PROGRAM PRG_Governance_Validator_Integrity_Governor
  VAR
    L_Now_MS : UDINT;
    L_Integrity_Valid : BOOL := TRUE;
    L_Error_Code : UDINT := 0;
    L_Error_Text : STRING(160) := '';
  END_VAR

            L_Now_MS := GVL_STATUS.G_System_Time_MS;
L_Integrity_Valid := TRUE;
L_Error_Code := 0;
L_Error_Text := '';

// Fail-safe defaults.
GVL_GOVERNANCE_VALIDATOR_INTEGRITY_FABRIC.Governance_Validator_Integrity_Valid := FALSE;
GVL_GOVERNANCE_VALIDATOR_INTEGRITY_FABRIC.Governance_Validator_Integrity_Granted := FALSE;
GVL_GOVERNANCE_VALIDATOR_INTEGRITY_FABRIC.Governance_Validator_Integrity_Quarantine_Active := TRUE;

GVL_GOVERNANCE_VALIDATOR_INTEGRITY_FABRIC.Validator_Semantics_Immutable := FALSE;
GVL_GOVERNANCE_VALIDATOR_INTEGRITY_FABRIC.CrossEpoch_Validation_Equivalence_Stable := FALSE;
GVL_GOVERNANCE_VALIDATOR_INTEGRITY_FABRIC.Distributed_Validator_Consensus_Valid := FALSE;
GVL_GOVERNANCE_VALIDATOR_INTEGRITY_FABRIC.Governance_Rule_Integrity_Canonical := FALSE;
GVL_GOVERNANCE_VALIDATOR_INTEGRITY_FABRIC.Validator_Lineage_Coherent := FALSE;

// Governance feedback integrity required.
IF NOT GVL_GOVERNANCE_FEEDBACK_INTEGRITY_FABRIC.Governance_Feedback_Integrity_Granted THEN
    L_Integrity_Valid := FALSE;
    L_Error_Code := 53000;
    L_Error_Text := 'Governance feedback integrity not granted';
END_IF;

// Validator self-corruption detectors.
IF GVL_GOVERNANCE_VALIDATOR_INTEGRITY_FABRIC.Validator_Semantic_Drift_Detected THEN
    L_Integrity_Valid := FALSE;
    L_Error_Code := 53001;
    L_Error_Text := 'Validator semantic drift detected';
END_IF;

IF GVL_GOVERNANCE_VALIDATOR_INTEGRITY_FABRIC.CrossNode_Validation_Fork THEN
    L_Integrity_Valid := FALSE;
    L_Error_Code := 53002;
    L_Error_Text := 'Cross-node validation fork detected';
END_IF;

IF GVL_GOVERNANCE_VALIDATOR_INTEGRITY_FABRIC.Governance_Rule_Mutation_Detected THEN
    L_Integrity_Valid := FALSE;
    L_Error_Code := 53003;
    L_Error_Text := 'Governance rule mutation detected';
END_IF;

IF GVL_GOVERNANCE_VALIDATOR_INTEGRITY_FABRIC.SelfReferential_Validator_Corruption THEN
    L_Integrity_Valid := FALSE;
    L_Error_Code := 53004;
    L_Error_Text := 'Self-referential validator corruption detected';
END_IF;

IF GVL_GOVERNANCE_VALIDATOR_INTEGRITY_FABRIC.Validator_Lineage_Drift_Detected THEN
    L_Integrity_Valid := FALSE;
    L_Error_Code := 53005;
    L_Error_Text := 'Validator lineage drift detected';
END_IF;

IF GVL_GOVERNANCE_VALIDATOR_INTEGRITY_FABRIC.Distributed_Validator_Reality_Fork_Detected THEN
    L_Integrity_Valid := FALSE;
    L_Error_Code := 53006;
    L_Error_Text := 'Distributed validator reality fork detected';
END_IF;

// Validator integrity validation.
IF L_Integrity_Valid
AND NOT GVL_GOVERNANCE_VALIDATOR_INTEGRITY_FABRIC.Validator_Causality_Grounded THEN
    L_Integrity_Valid := FALSE;
    L_Error_Code := 53010;
    L_Error_Text := 'Validator causality invalid';
END_IF;

IF L_Integrity_Valid
AND NOT GVL_GOVERNANCE_VALIDATOR_INTEGRITY_FABRIC.Governance_Rule_Evolution_Governed THEN
    L_Integrity_Valid := FALSE;
    L_Error_Code := 53011;
    L_Error_Text := 'Governance rule evolution invalid';
END_IF;

IF L_Integrity_Valid
AND NOT GVL_GOVERNANCE_VALIDATOR_INTEGRITY_FABRIC.Distributed_Validation_Timeline_Monotonic THEN
    L_Integrity_Valid := FALSE;
    L_Error_Code := 53012;
    L_Error_Text := 'Distributed validation timeline monotonicity invalid';
END_IF;

IF L_Integrity_Valid
AND NOT GVL_GOVERNANCE_VALIDATOR_INTEGRITY_FABRIC.Validator_Interpretation_Equivalence_Valid THEN
    L_Integrity_Valid := FALSE;
    L_Error_Code := 53013;
    L_Error_Text := 'Validator interpretation equivalence invalid';
END_IF;

IF L_Integrity_Valid THEN
    GVL_GOVERNANCE_VALIDATOR_INTEGRITY_FABRIC.Governance_Validator_Integrity_Valid := TRUE;
    GVL_GOVERNANCE_VALIDATOR_INTEGRITY_FABRIC.Governance_Validator_Integrity_Granted := TRUE;
    GVL_GOVERNANCE_VALIDATOR_INTEGRITY_FABRIC.Governance_Validator_Integrity_Quarantine_Active := FALSE;

    GVL_GOVERNANCE_VALIDATOR_INTEGRITY_FABRIC.Validator_Semantics_Immutable := TRUE;
    GVL_GOVERNANCE_VALIDATOR_INTEGRITY_FABRIC.CrossEpoch_Validation_Equivalence_Stable := TRUE;
    GVL_GOVERNANCE_VALIDATOR_INTEGRITY_FABRIC.Distributed_Validator_Consensus_Valid := TRUE;
    GVL_GOVERNANCE_VALIDATOR_INTEGRITY_FABRIC.Governance_Rule_Integrity_Canonical := TRUE;
    GVL_GOVERNANCE_VALIDATOR_INTEGRITY_FABRIC.Validator_Lineage_Coherent := TRUE;

    GVL_GOVERNANCE_VALIDATOR_INTEGRITY_FABRIC.Governance_Validator_Integrity_Epoch :=
        GVL_GOVERNANCE_FEEDBACK_INTEGRITY_FABRIC.Governance_Feedback_Integrity_Epoch;

    GVL_GOVERNANCE_VALIDATOR_INTEGRITY_FABRIC.Governance_Validator_Integrity_Epoch_Coherent := TRUE;

    GVL_GOVERNANCE_VALIDATOR_INTEGRITY_FABRIC.Governance_Validator_Integrity_Last_Update_MS :=
        L_Now_MS;

    GVL_GOVERNANCE_VALIDATOR_INTEGRITY_FABRIC.Governance_Validator_Integrity_Lease_Expired := FALSE;

    GVL_GOVERNANCE_VALIDATOR_INTEGRITY_FABRIC.Governance_Validator_Integrity_Last_Error_Code := 0;
    GVL_GOVERNANCE_VALIDATOR_INTEGRITY_FABRIC.Governance_Validator_Integrity_Last_Error_Text := '';
ELSE
    GVL_GOVERNANCE_VALIDATOR_INTEGRITY_FABRIC.Governance_Validator_Integrity_Valid := FALSE;
    GVL_GOVERNANCE_VALIDATOR_INTEGRITY_FABRIC.Governance_Validator_Integrity_Granted := FALSE;
    GVL_GOVERNANCE_VALIDATOR_INTEGRITY_FABRIC.Governance_Validator_Integrity_Quarantine_Active := TRUE;

    GVL_GOVERNANCE_VALIDATOR_INTEGRITY_FABRIC.Governance_Validator_Integrity_Lease_Expired := TRUE;

    GVL_GOVERNANCE_VALIDATOR_INTEGRITY_FABRIC.Governance_Validator_Integrity_Last_Error_Code :=
        L_Error_Code;

    GVL_GOVERNANCE_VALIDATOR_INTEGRITY_FABRIC.Governance_Validator_Integrity_Last_Error_Text :=
        L_Error_Text;

    GVL_GOVERNANCE_VALIDATOR_INTEGRITY_FABRIC.Governance_Validator_Integrity_Invalidation_Count :=
        GVL_GOVERNANCE_VALIDATOR_INTEGRITY_FABRIC.Governance_Validator_Integrity_Invalidation_Count + 1;
END_IF;
          
END_PROGRAM

PROGRAM PRG_Heating_Policy_Observer
  VAR
    fbPolicy : FB_Heating_Policy_Observer;
  END_VAR

            fbPolicy(
    VI_Zone_Occupied := GVL_PRESENCE.G_Zone_Occupied,
    VI_Zone_Last_Motion_TS := GVL_PRESENCE.G_Zone_Last_Motion_TS,
    VI_System_Time_MS := GVL_STATUS.G_System_Time_MS,
    VI_Zone_Permanent_Use := GVL_HEATING_POLICY.G_Zone_Permanent_Use,
    VI_Zone_Guest_Preheat := GVL_HEATING_POLICY.G_Zone_Guest_Preheat_Request,
    VI_Behavior_Mode := GVL_MODE.G_Current_Behavior_Mode
);

GVL_HEATING_POLICY.G_Zone_Empty_Duration_MS := fbPolicy.VO_Zone_Empty_Duration_MS;
GVL_HEATING_POLICY.G_Zone_Policy_Class := fbPolicy.VO_Zone_Policy_Class;
GVL_HEATING_POLICY.G_Zone_Target_Adjustment := fbPolicy.VO_Zone_Target_Adjustment;
GVL_HEATING_POLICY.G_Zone_Priority_Bias := fbPolicy.VO_Zone_Priority_Bias;
          
END_PROGRAM

PROGRAM PRG_Time_Service
  VAR
    fbTimebase : FB_System_Timebase;
    fbTime : FB_Time_Service;
  END_VAR

            // Central time update point.
// Must run before PRG_IO_Read and all consumers of GVL_TIME_SERVICE.
fbTimebase();
fbTime();

// Step 4.2 compatibility bridge.
// Legacy consumers of GVL_STATUS.G_System_Time_MS receive the same canonical time.
GVL_STATUS.G_System_Time_MS := GVL_TIME_SERVICE.G_Now_MS;
GVL_STATUS.G_Current_TOD := GVL_TIME_SERVICE.G_Current_TOD;
GVL_STATUS.G_Current_Day := TO_UINT(GVL_TIME_SERVICE.G_Day_Of_Week);
          
END_PROGRAM

PROGRAM PRG_Operator_Semantic_Alignment_Governor
  VAR
    L_Now_MS : UDINT;
    L_Operator_Valid : BOOL := TRUE;
    L_Error_Code : UDINT := 0;
    L_Error_Text : STRING(160) := '';
  END_VAR

            L_Now_MS := GVL_STATUS.G_System_Time_MS;
L_Operator_Valid := TRUE;
L_Error_Code := 0;
L_Error_Text := '';

// Fail-safe defaults.
GVL_OPERATOR_SEMANTIC_ALIGNMENT.Operator_Semantic_Alignment_Valid := FALSE;
GVL_OPERATOR_SEMANTIC_ALIGNMENT.Operator_Semantic_Alignment_Granted := FALSE;
GVL_OPERATOR_SEMANTIC_ALIGNMENT.Operator_Semantic_Alignment_Quarantine_Active := TRUE;

GVL_OPERATOR_SEMANTIC_ALIGNMENT.HMI_Semantic_State_Coherent := FALSE;
GVL_OPERATOR_SEMANTIC_ALIGNMENT.Operator_Recovery_Intent_Aligned := FALSE;
GVL_OPERATOR_SEMANTIC_ALIGNMENT.Alarm_Semantic_Priority_Coherent := FALSE;
GVL_OPERATOR_SEMANTIC_ALIGNMENT.Runtime_Explanation_Coherent := FALSE;
GVL_OPERATOR_SEMANTIC_ALIGNMENT.Authority_State_Human_Visible := FALSE;

// Semantic preservation required.
IF NOT GVL_SEMANTIC_PRESERVATION_FABRIC.Semantic_Preservation_Granted THEN
    L_Operator_Valid := FALSE;
    L_Error_Code := 40000;
    L_Error_Text := 'Semantic preservation authority not granted';
END_IF;

// Human-machine semantic split-brain detectors.
IF GVL_OPERATOR_SEMANTIC_ALIGNMENT.HMI_Semantic_Lag_Detected THEN
    L_Operator_Valid := FALSE;
    L_Error_Code := 40001;
    L_Error_Text := 'HMI semantic lag detected';
END_IF;

IF GVL_OPERATOR_SEMANTIC_ALIGNMENT.Operator_Interpretation_Skew_Detected THEN
    L_Operator_Valid := FALSE;
    L_Error_Code := 40002;
    L_Error_Text := 'Operator interpretation skew detected';
END_IF;

IF GVL_OPERATOR_SEMANTIC_ALIGNMENT.Alarm_Cognition_Mismatch_Detected THEN
    L_Operator_Valid := FALSE;
    L_Error_Code := 40003;
    L_Error_Text := 'Alarm cognition mismatch detected';
END_IF;

IF GVL_OPERATOR_SEMANTIC_ALIGNMENT.Hidden_Authority_State_Detected THEN
    L_Operator_Valid := FALSE;
    L_Error_Code := 40004;
    L_Error_Text := 'Hidden authority state detected';
END_IF;

IF GVL_OPERATOR_SEMANTIC_ALIGNMENT.Semantic_Explanation_Divergence_Detected THEN
    L_Operator_Valid := FALSE;
    L_Error_Code := 40005;
    L_Error_Text := 'Semantic explanation divergence detected';
END_IF;

IF GVL_OPERATOR_SEMANTIC_ALIGNMENT.Human_Recovery_Misunderstanding_Detected THEN
    L_Operator_Valid := FALSE;
    L_Error_Code := 40006;
    L_Error_Text := 'Human recovery misunderstanding detected';
END_IF;

// Operator cognition coherence validation.
IF L_Operator_Valid
AND NOT GVL_OPERATOR_SEMANTIC_ALIGNMENT.Human_Interpretation_Coherent THEN
    L_Operator_Valid := FALSE;
    L_Error_Code := 40010;
    L_Error_Text := 'Human interpretation coherence invalid';
END_IF;

IF L_Operator_Valid
AND NOT GVL_OPERATOR_SEMANTIC_ALIGNMENT.Adaptive_Runtime_Visibility_Valid THEN
    L_Operator_Valid := FALSE;
    L_Error_Code := 40011;
    L_Error_Text := 'Adaptive runtime visibility invalid';
END_IF;

IF L_Operator_Valid
AND NOT GVL_OPERATOR_SEMANTIC_ALIGNMENT.Semantic_Explanation_Fresh THEN
    L_Operator_Valid := FALSE;
    L_Error_Code := 40012;
    L_Error_Text := 'Semantic explanation freshness invalid';
END_IF;

IF L_Operator_Valid
AND NOT GVL_OPERATOR_SEMANTIC_ALIGNMENT.Operator_Action_Context_Aligned THEN
    L_Operator_Valid := FALSE;
    L_Error_Code := 40013;
    L_Error_Text := 'Operator action context alignment invalid';
END_IF;

IF L_Operator_Valid THEN
    GVL_OPERATOR_SEMANTIC_ALIGNMENT.Operator_Semantic_Alignment_Valid := TRUE;
    GVL_OPERATOR_SEMANTIC_ALIGNMENT.Operator_Semantic_Alignment_Granted := TRUE;
    GVL_OPERATOR_SEMANTIC_ALIGNMENT.Operator_Semantic_Alignment_Quarantine_Active := FALSE;

    GVL_OPERATOR_SEMANTIC_ALIGNMENT.HMI_Semantic_State_Coherent := TRUE;
    GVL_OPERATOR_SEMANTIC_ALIGNMENT.Operator_Recovery_Intent_Aligned := TRUE;
    GVL_OPERATOR_SEMANTIC_ALIGNMENT.Alarm_Semantic_Priority_Coherent := TRUE;
    GVL_OPERATOR_SEMANTIC_ALIGNMENT.Runtime_Explanation_Coherent := TRUE;
    GVL_OPERATOR_SEMANTIC_ALIGNMENT.Authority_State_Human_Visible := TRUE;

    GVL_OPERATOR_SEMANTIC_ALIGNMENT.Operator_Alignment_Epoch :=
        GVL_SEMANTIC_PRESERVATION_FABRIC.Semantic_Preservation_Epoch;

    GVL_OPERATOR_SEMANTIC_ALIGNMENT.Operator_Alignment_Epoch_Coherent := TRUE;

    GVL_OPERATOR_SEMANTIC_ALIGNMENT.Operator_Alignment_Last_Update_MS :=
        L_Now_MS;

    GVL_OPERATOR_SEMANTIC_ALIGNMENT.Operator_Alignment_Lease_Expired := FALSE;

    GVL_OPERATOR_SEMANTIC_ALIGNMENT.Operator_Alignment_Last_Error_Code := 0;
    GVL_OPERATOR_SEMANTIC_ALIGNMENT.Operator_Alignment_Last_Error_Text := '';
ELSE
    GVL_OPERATOR_SEMANTIC_ALIGNMENT.Operator_Semantic_Alignment_Valid := FALSE;
    GVL_OPERATOR_SEMANTIC_ALIGNMENT.Operator_Semantic_Alignment_Granted := FALSE;
    GVL_OPERATOR_SEMANTIC_ALIGNMENT.Operator_Semantic_Alignment_Quarantine_Active := TRUE;

    GVL_OPERATOR_SEMANTIC_ALIGNMENT.Operator_Alignment_Lease_Expired := TRUE;

    GVL_OPERATOR_SEMANTIC_ALIGNMENT.Operator_Alignment_Last_Error_Code :=
        L_Error_Code;

    GVL_OPERATOR_SEMANTIC_ALIGNMENT.Operator_Alignment_Last_Error_Text :=
        L_Error_Text;

    GVL_OPERATOR_SEMANTIC_ALIGNMENT.Operator_Alignment_Invalidation_Count :=
        GVL_OPERATOR_SEMANTIC_ALIGNMENT.Operator_Alignment_Invalidation_Count + 1;
END_IF;
          
END_PROGRAM

PROGRAM PRG_Deterministic_Recovery_Path_Governor
  VAR
    L_Now_MS : UDINT;
  END_VAR

            L_Now_MS := GVL_STATUS.G_System_Time_MS;

IF GVL_CROSSDOMAIN_FAILSAFE_CLOSURE_FABRIC.CrossDomain_FailSafe_Closure_Granted
AND NOT GVL_DETERMINISTIC_RECOVERY_PATH_FABRIC.Unsafe_Recovery_Path_Detected
AND NOT GVL_DETERMINISTIC_RECOVERY_PATH_FABRIC.Recovery_Path_Divergence_Detected
AND NOT GVL_DETERMINISTIC_RECOVERY_PATH_FABRIC.Recovery_Causality_Break_Detected
AND NOT GVL_DETERMINISTIC_RECOVERY_PATH_FABRIC.Distributed_Recovery_Fork_Detected THEN

    GVL_DETERMINISTIC_RECOVERY_PATH_FABRIC.Deterministic_Recovery_Path_Valid := TRUE;
    GVL_DETERMINISTIC_RECOVERY_PATH_FABRIC.Deterministic_Recovery_Path_Granted := TRUE;
    GVL_DETERMINISTIC_RECOVERY_PATH_FABRIC.Deterministic_Recovery_Path_Canonical := TRUE;
    GVL_DETERMINISTIC_RECOVERY_PATH_FABRIC.Recovery_Lineage_Causality_Valid := TRUE;
    GVL_DETERMINISTIC_RECOVERY_PATH_FABRIC.Recovery_Physical_Convergence_Stable := TRUE;
    GVL_DETERMINISTIC_RECOVERY_PATH_FABRIC.Recovery_Timeline_Monotonic := TRUE;

    GVL_DETERMINISTIC_RECOVERY_PATH_FABRIC.Deterministic_Recovery_Path_Epoch :=
        GVL_CROSSDOMAIN_FAILSAFE_CLOSURE_FABRIC.CrossDomain_FailSafe_Closure_Epoch;

    GVL_DETERMINISTIC_RECOVERY_PATH_FABRIC.Deterministic_Recovery_Path_Last_Update_MS :=
        L_Now_MS;
END_IF;
          
END_PROGRAM

PROGRAM PRG_Temporal_Causality_Closure_Governor

            IF GVL_DISTRIBUTED_SAFETY_REALITY_CONSENSUS_FABRIC.Distributed_Safety_Reality_Consensus_Granted
AND NOT GVL_TEMPORAL_CAUSALITY_CLOSURE_FABRIC.Temporal_Fork_Detected
AND NOT GVL_TEMPORAL_CAUSALITY_CLOSURE_FABRIC.Stale_Causality_Application_Detected
AND NOT GVL_TEMPORAL_CAUSALITY_CLOSURE_FABRIC.Recovery_Before_Revocation_Detected
AND NOT GVL_TEMPORAL_CAUSALITY_CLOSURE_FABRIC.Distributed_Timeline_Drift_Detected THEN

    GVL_TEMPORAL_CAUSALITY_CLOSURE_FABRIC.Temporal_Causality_Closure_Valid := TRUE;
    GVL_TEMPORAL_CAUSALITY_CLOSURE_FABRIC.Temporal_Causality_Closure_Granted := TRUE;
    GVL_TEMPORAL_CAUSALITY_CLOSURE_FABRIC.Temporal_Causality_Coherent := TRUE;
    GVL_TEMPORAL_CAUSALITY_CLOSURE_FABRIC.Monotonic_Reality_Timeline_Valid := TRUE;
    GVL_TEMPORAL_CAUSALITY_CLOSURE_FABRIC.Recovery_Revocation_Ordering_Valid := TRUE;
END_IF;
          
END_PROGRAM

PROGRAM PRG_Governance_Liveness_Integrity_Governor
  VAR
    L_Now_MS : UDINT;
    L_Integrity_Valid : BOOL := TRUE;
    L_Error_Code : UDINT := 0;
    L_Error_Text : STRING(160) := '';
  END_VAR

            L_Now_MS := GVL_STATUS.G_System_Time_MS;
L_Integrity_Valid := TRUE;
L_Error_Code := 0;
L_Error_Text := '';

// Fail-safe defaults.
GVL_GOVERNANCE_LIVENESS_INTEGRITY_FABRIC.Governance_Liveness_Integrity_Valid := FALSE;
GVL_GOVERNANCE_LIVENESS_INTEGRITY_FABRIC.Governance_Liveness_Integrity_Granted := FALSE;
GVL_GOVERNANCE_LIVENESS_INTEGRITY_FABRIC.Governance_Liveness_Integrity_Quarantine_Active := TRUE;

GVL_GOVERNANCE_LIVENESS_INTEGRITY_FABRIC.Governance_Execution_Liveness_Stable := FALSE;
GVL_GOVERNANCE_LIVENESS_INTEGRITY_FABRIC.Integrity_Governor_Scheduling_Canonical := FALSE;
GVL_GOVERNANCE_LIVENESS_INTEGRITY_FABRIC.CrossGovernor_Execution_Continuity_Valid := FALSE;
GVL_GOVERNANCE_LIVENESS_INTEGRITY_FABRIC.Deterministic_Validation_Cycle_Integrity := FALSE;
GVL_GOVERNANCE_LIVENESS_INTEGRITY_FABRIC.Governance_Runtime_Liveness_Coherent := FALSE;

// Governance validator integrity required.
IF NOT GVL_GOVERNANCE_VALIDATOR_INTEGRITY_FABRIC.Governance_Validator_Integrity_Granted THEN
    L_Integrity_Valid := FALSE;
    L_Error_Code := 54000;
    L_Error_Text := 'Governance validator integrity not granted';
END_IF;

// Governance liveness degradation detectors.
IF GVL_GOVERNANCE_LIVENESS_INTEGRITY_FABRIC.Integrity_Governor_Starvation_Detected THEN
    L_Integrity_Valid := FALSE;
    L_Error_Code := 54001;
    L_Error_Text := 'Integrity governor starvation detected';
END_IF;

IF GVL_GOVERNANCE_LIVENESS_INTEGRITY_FABRIC.Validation_Cycle_Skip_Detected THEN
    L_Integrity_Valid := FALSE;
    L_Error_Code := 54002;
    L_Error_Text := 'Validation cycle skip detected';
END_IF;

IF GVL_GOVERNANCE_LIVENESS_INTEGRITY_FABRIC.CrossGovernor_Execution_Jitter_Fork THEN
    L_Integrity_Valid := FALSE;
    L_Error_Code := 54003;
    L_Error_Text := 'Cross-governor execution jitter fork detected';
END_IF;

IF GVL_GOVERNANCE_LIVENESS_INTEGRITY_FABRIC.Selective_Governance_Degradation_Detected THEN
    L_Integrity_Valid := FALSE;
    L_Error_Code := 54004;
    L_Error_Text := 'Selective governance degradation detected';
END_IF;

IF GVL_GOVERNANCE_LIVENESS_INTEGRITY_FABRIC.Runtime_Governor_Execution_Stall_Detected THEN
    L_Integrity_Valid := FALSE;
    L_Error_Code := 54005;
    L_Error_Text := 'Runtime governor execution stall detected';
END_IF;

IF GVL_GOVERNANCE_LIVENESS_INTEGRITY_FABRIC.Distributed_Liveness_Reality_Fork_Detected THEN
    L_Integrity_Valid := FALSE;
    L_Error_Code := 54006;
    L_Error_Text := 'Distributed liveness reality fork detected';
END_IF;

// Governance liveness validation.
IF L_Integrity_Valid
AND NOT GVL_GOVERNANCE_LIVENESS_INTEGRITY_FABRIC.Validation_Cycle_Timing_Monotonic THEN
    L_Integrity_Valid := FALSE;
    L_Error_Code := 54010;
    L_Error_Text := 'Validation cycle timing invalid';
END_IF;

IF L_Integrity_Valid
AND NOT GVL_GOVERNANCE_LIVENESS_INTEGRITY_FABRIC.Distributed_Governor_Execution_Aligned THEN
    L_Integrity_Valid := FALSE;
    L_Error_Code := 54011;
    L_Error_Text := 'Distributed governor execution alignment invalid';
END_IF;

IF L_Integrity_Valid
AND NOT GVL_GOVERNANCE_LIVENESS_INTEGRITY_FABRIC.Runtime_Integrity_Causality_Grounded THEN
    L_Integrity_Valid := FALSE;
    L_Error_Code := 54012;
    L_Error_Text := 'Runtime integrity causality invalid';
END_IF;

IF L_Integrity_Valid
AND NOT GVL_GOVERNANCE_LIVENESS_INTEGRITY_FABRIC.Governance_Execution_Budget_Stable THEN
    L_Integrity_Valid := FALSE;
    L_Error_Code := 54013;
    L_Error_Text := 'Governance execution budget invalid';
END_IF;

IF L_Integrity_Valid THEN
    GVL_GOVERNANCE_LIVENESS_INTEGRITY_FABRIC.Governance_Liveness_Integrity_Valid := TRUE;
    GVL_GOVERNANCE_LIVENESS_INTEGRITY_FABRIC.Governance_Liveness_Integrity_Granted := TRUE;
    GVL_GOVERNANCE_LIVENESS_INTEGRITY_FABRIC.Governance_Liveness_Integrity_Quarantine_Active := FALSE;

    GVL_GOVERNANCE_LIVENESS_INTEGRITY_FABRIC.Governance_Execution_Liveness_Stable := TRUE;
    GVL_GOVERNANCE_LIVENESS_INTEGRITY_FABRIC.Integrity_Governor_Scheduling_Canonical := TRUE;
    GVL_GOVERNANCE_LIVENESS_INTEGRITY_FABRIC.CrossGovernor_Execution_Continuity_Valid := TRUE;
    GVL_GOVERNANCE_LIVENESS_INTEGRITY_FABRIC.Deterministic_Validation_Cycle_Integrity := TRUE;
    GVL_GOVERNANCE_LIVENESS_INTEGRITY_FABRIC.Governance_Runtime_Liveness_Coherent := TRUE;

    GVL_GOVERNANCE_LIVENESS_INTEGRITY_FABRIC.Governance_Liveness_Integrity_Epoch :=
        GVL_GOVERNANCE_VALIDATOR_INTEGRITY_FABRIC.Governance_Validator_Integrity_Epoch;

    GVL_GOVERNANCE_LIVENESS_INTEGRITY_FABRIC.Governance_Liveness_Integrity_Epoch_Coherent := TRUE;

    GVL_GOVERNANCE_LIVENESS_INTEGRITY_FABRIC.Governance_Liveness_Integrity_Last_Update_MS :=
        L_Now_MS;

    GVL_GOVERNANCE_LIVENESS_INTEGRITY_FABRIC.Governance_Liveness_Integrity_Lease_Expired := FALSE;

    GVL_GOVERNANCE_LIVENESS_INTEGRITY_FABRIC.Governance_Liveness_Integrity_Last_Error_Code := 0;
    GVL_GOVERNANCE_LIVENESS_INTEGRITY_FABRIC.Governance_Liveness_Integrity_Last_Error_Text := '';
ELSE
    GVL_GOVERNANCE_LIVENESS_INTEGRITY_FABRIC.Governance_Liveness_Integrity_Valid := FALSE;
    GVL_GOVERNANCE_LIVENESS_INTEGRITY_FABRIC.Governance_Liveness_Integrity_Granted := FALSE;
    GVL_GOVERNANCE_LIVENESS_INTEGRITY_FABRIC.Governance_Liveness_Integrity_Quarantine_Active := TRUE;

    GVL_GOVERNANCE_LIVENESS_INTEGRITY_FABRIC.Governance_Liveness_Integrity_Lease_Expired := TRUE;

    GVL_GOVERNANCE_LIVENESS_INTEGRITY_FABRIC.Governance_Liveness_Integrity_Last_Error_Code :=
        L_Error_Code;

    GVL_GOVERNANCE_LIVENESS_INTEGRITY_FABRIC.Governance_Liveness_Integrity_Last_Error_Text :=
        L_Error_Text;

    GVL_GOVERNANCE_LIVENESS_INTEGRITY_FABRIC.Governance_Liveness_Integrity_Invalidation_Count :=
        GVL_GOVERNANCE_LIVENESS_INTEGRITY_FABRIC.Governance_Liveness_Integrity_Invalidation_Count + 1;
END_IF;
          
END_PROGRAM

PROGRAM PRG_Runtime_Compression_Governor

            // ARCHITECTURAL CONSOLIDATION & RUNTIME COMPRESSION
// READ-ONLY / NON-INVASIVE

GVL_CANONICAL_RUNTIME_FABRIC_REGISTRY.Runtime_Complexity_Pressure_Observed :=
    GVL_SURVIVABILITY_INTELLIGENCE_FABRIC.Governance_Saturation_Pressure_Observed;

GVL_CANONICAL_RUNTIME_FABRIC_REGISTRY.Governance_Runtime_Cost_Observed :=
    GVL_OPERATIONAL_INTELLIGENCE_FABRIC.Governance_Complexity_Pressure_Observed;

GVL_CANONICAL_RUNTIME_FABRIC_REGISTRY.Verification_Induced_Instability_Risk :=
    GVL_SURVIVABILITY_INTELLIGENCE_FABRIC.Chronic_Degradation_Risk_Increasing;

IF GVL_OPERATIONAL_INTELLIGENCE_FABRIC.Governance_Saturation_Observed THEN
    GVL_CANONICAL_RUNTIME_FABRIC_REGISTRY.Governance_Scattering_Observed := TRUE;
    GVL_CANONICAL_RUNTIME_FABRIC_REGISTRY.Semantic_Duplication_Observed := TRUE;
END_IF;

IF GVL_CANONICAL_RUNTIME_FABRIC_REGISTRY.Runtime_Complexity_Pressure_Observed THEN
    GVL_CANONICAL_RUNTIME_FABRIC_REGISTRY.Governance_Depth_Limit_Reached := TRUE;
END_IF;

IF GVL_CANONICAL_RUNTIME_FABRIC_REGISTRY.Governance_Runtime_Cost_Observed THEN
    GVL_CANONICAL_RUNTIME_FABRIC_REGISTRY.Verification_Chaining_Limit_Reached := TRUE;
END_IF;

IF GVL_OPERATIONAL_INTELLIGENCE_FABRIC.Operational_Opacity_Observed THEN
    GVL_CANONICAL_RUNTIME_FABRIC_REGISTRY.Observability_Amplification_Limit_Reached := TRUE;
END_IF;
          
END_PROGRAM

PROGRAM PRG_Distributed_Runtime_Supervisor
  VAR
    fbClusterSafetyBarrier : FB_Cluster_Safety_Barrier_Runtime;
    fbRuntimeDiscovery : FB_Runtime_Node_Discovery;
    fbRuntimeSessions : FB_Runtime_Session_Governance;
    fbDistributedRuntimeContinuity : FB_Distributed_Runtime_Continuity;
    fbDistributedAuthority : FB_Distributed_Authority_Arbitration;
    fbRuntimeBusReplication : FB_Runtime_Bus_Replication;
    fbMQTTRuntimeAdapter : FB_MQTT_Runtime_Adapter;
    fbOPCUARuntimeAdapter : FB_OPCUA_Runtime_Adapter;
    fbADSRuntimeAdapter : FB_ADS_Runtime_Adapter;
    fbProjectionOwnership : FB_Distributed_Projection_Ownership_Runtime;
    fbDistributedOrchestration : FB_Distributed_Orchestration_Runtime;
    fbRecoveryLock : FB_Distributed_Recovery_Lock_Runtime;
    fbExecutionGates : FB_Distributed_Execution_Gates_Runtime;
    fbClusterRuntimeFSM : FB_Cluster_Runtime_FSM;
  END_VAR

            // Root distributed runtime execution chain.
//
// Execution order intentionally deterministic:
// safety -> discovery -> sessions -> authority -> replication
// -> transport -> ownership -> orchestration -> recovery locking
// -> unified execution gates -> cluster runtime FSM.
//
// Important convergence contract:
// execution gates must never reopen distributed execution authority
// before finalized convergence/publication continuity is achieved.
//
// Required finalized authority chain:
// immutable snapshot
// -> distributed reconciliation
// -> distributed commit continuity
// -> finalized publication validity
// -> convergence release
// -> execution gates reopen.

fbClusterSafetyBarrier(
    VI_Enable := TRUE,
    VI_System_Time_MS := GVL_STATUS.G_System_Time_MS
);

fbRuntimeDiscovery(
    VI_Enable := TRUE,
    VI_System_Time_MS := GVL_STATUS.G_System_Time_MS
);

fbRuntimeSessions(
    VI_Enable := TRUE,
    VI_System_Time_MS := GVL_STATUS.G_System_Time_MS
);

fbDistributedRuntimeContinuity(
    VI_Enable := TRUE,
    VI_System_Time_MS := GVL_STATUS.G_System_Time_MS
);

fbDistributedAuthority(
    VI_Enable := TRUE,
    VI_System_Time_MS := GVL_STATUS.G_System_Time_MS
);

fbRuntimeBusReplication(
    VI_Enable := TRUE,
    VI_System_Time_MS := GVL_STATUS.G_System_Time_MS
);

fbMQTTRuntimeAdapter(
    VI_Enable := TRUE,
    VI_System_Time_MS := GVL_STATUS.G_System_Time_MS
);

fbOPCUARuntimeAdapter(
    VI_Enable := TRUE,
    VI_System_Time_MS := GVL_STATUS.G_System_Time_MS
);

fbADSRuntimeAdapter(
    VI_Enable := TRUE,
    VI_System_Time_MS := GVL_STATUS.G_System_Time_MS
);

fbProjectionOwnership(
    VI_Enable := TRUE,
    VI_System_Time_MS := GVL_STATUS.G_System_Time_MS
);

fbDistributedOrchestration(
    VI_Enable := TRUE,
    VI_System_Time_MS := GVL_STATUS.G_System_Time_MS
);

fbRecoveryLock(
    VI_Enable := TRUE,
    VI_System_Time_MS := GVL_STATUS.G_System_Time_MS
);

fbExecutionGates(
    VI_Enable := TRUE,
    VI_System_Time_MS := GVL_STATUS.G_System_Time_MS
);

fbClusterRuntimeFSM(
    VI_Enable := TRUE,
    VI_System_Time_MS := GVL_STATUS.G_System_Time_MS
);
          
END_PROGRAM

PROGRAM PRG_Authority_Lineage_Governor
  VAR
    L_Now_MS : UDINT;
    L_Lineage_Valid : BOOL := TRUE;
    L_Error_Code : UDINT := 0;
    L_Error_Text : STRING(160) := '';
  END_VAR

            L_Now_MS := GVL_STATUS.G_System_Time_MS;
L_Lineage_Valid := TRUE;
L_Error_Code := 0;
L_Error_Text := '';

GVL_AUTHORITY_LINEAGE.Authority_Lineage_Valid := FALSE;
GVL_AUTHORITY_LINEAGE.Warm_Restart_Continuity_Valid := FALSE;
GVL_AUTHORITY_LINEAGE.HA_Resume_Continuity_Valid := FALSE;
GVL_AUTHORITY_LINEAGE.Retained_State_Integrity_Valid := FALSE;

IF GVL_AUTHORITY_LINEAGE.Authority_Replay_Suspected THEN
    L_Lineage_Valid := FALSE;
    L_Error_Code := 25000;
    L_Error_Text := 'Authority replay suspected';
END_IF;

IF L_Lineage_Valid AND GVL_AUTHORITY_LINEAGE.Retained_State_Skew_Detected THEN
    L_Lineage_Valid := FALSE;
    L_Error_Code := 25001;
    L_Error_Text := 'Retained state skew detected';
END_IF;

IF L_Lineage_Valid AND GVL_AUTHORITY_LINEAGE.Partial_Authority_Resurrection_Detected THEN
    L_Lineage_Valid := FALSE;
    L_Error_Code := 25002;
    L_Error_Text := 'Partial authority resurrection detected';
END_IF;

IF L_Lineage_Valid AND GVL_AUTHORITY_LINEAGE.Epoch_Lineage_Discontinuity_Detected THEN
    L_Lineage_Valid := FALSE;
    L_Error_Code := 25003;
    L_Error_Text := 'Epoch lineage discontinuity detected';
END_IF;

IF L_Lineage_Valid
AND (ULINT_TO_UDINT(GVL_PHYSICAL_AUTHORITY_EPOCH.Physical_Authority_Epoch) < GVL_AUTHORITY_LINEAGE.Last_Physical_Authority_Epoch) THEN
    GVL_AUTHORITY_LINEAGE.Authority_Replay_Suspected := TRUE;
    L_Lineage_Valid := FALSE;
    L_Error_Code := 25010;
    L_Error_Text := 'Physical authority epoch rollback detected';
END_IF;

IF L_Lineage_Valid
AND (ULINT_TO_UDINT(GVL_RUNTIME_EPOCH.Runtime_Epoch) < GVL_AUTHORITY_LINEAGE.Last_Runtime_Epoch) THEN
    GVL_AUTHORITY_LINEAGE.Retained_State_Skew_Detected := TRUE;
    L_Lineage_Valid := FALSE;
    L_Error_Code := 25011;
    L_Error_Text := 'Runtime epoch rollback detected';
END_IF;

IF L_Lineage_Valid
AND (ULINT_TO_UDINT(GVL_OUTPUT_EPOCH.Output_Publication_Epoch) < GVL_AUTHORITY_LINEAGE.Last_Output_Publication_Epoch) THEN
    GVL_AUTHORITY_LINEAGE.Partial_Authority_Resurrection_Detected := TRUE;
    L_Lineage_Valid := FALSE;
    L_Error_Code := 25012;
    L_Error_Text := 'Output publication epoch rollback detected';
END_IF;

IF L_Lineage_Valid THEN
    GVL_AUTHORITY_LINEAGE.Authority_Lineage_Valid := TRUE;
    GVL_AUTHORITY_LINEAGE.Warm_Restart_Continuity_Valid := TRUE;
    GVL_AUTHORITY_LINEAGE.HA_Resume_Continuity_Valid := TRUE;
    GVL_AUTHORITY_LINEAGE.Retained_State_Integrity_Valid := TRUE;

    GVL_AUTHORITY_LINEAGE.Authority_Lineage_Epoch := ULINT_TO_UDINT(GVL_PHYSICAL_AUTHORITY_EPOCH.Physical_Authority_Epoch);
    GVL_AUTHORITY_LINEAGE.Last_Physical_Authority_Epoch := ULINT_TO_UDINT(GVL_PHYSICAL_AUTHORITY_EPOCH.Physical_Authority_Epoch);
    GVL_AUTHORITY_LINEAGE.Last_Runtime_Epoch := ULINT_TO_UDINT(GVL_RUNTIME_EPOCH.Runtime_Epoch);
    GVL_AUTHORITY_LINEAGE.Last_Output_Publication_Epoch := ULINT_TO_UDINT(GVL_OUTPUT_EPOCH.Output_Publication_Epoch);
    GVL_AUTHORITY_LINEAGE.Authority_Lineage_Last_Update_MS := L_Now_MS;
    GVL_AUTHORITY_LINEAGE.Authority_Lineage_Last_Error_Code := 0;
    GVL_AUTHORITY_LINEAGE.Authority_Lineage_Last_Error_Text := '';
ELSE
    GVL_AUTHORITY_LINEAGE.Authority_Lineage_Valid := FALSE;
    GVL_AUTHORITY_LINEAGE.Authority_Lineage_Last_Error_Code := L_Error_Code;
    GVL_AUTHORITY_LINEAGE.Authority_Lineage_Last_Error_Text := L_Error_Text;
    GVL_AUTHORITY_LINEAGE.Authority_Lineage_Invalidation_Count := GVL_AUTHORITY_LINEAGE.Authority_Lineage_Invalidation_Count + 1;
END_IF;
          
END_PROGRAM

PROGRAM PRG_System_Alarm_Gateway
  VAR
    fbSystemAlarmOrchestrator : FB_System_Alarm_Orchestrator;
    fbSystemGatewayIntent : FB_System_Gateway_Intent;
    L_Scenario_Req_Gateway : E_SCENARIO_TYPE;
  END_VAR

            // Alarm orchestration based on global health snapshot
fbSystemAlarmOrchestrator(
    VI_First_Fault_Active := GVL_SYSTEM_HEALTH.G_First_Fault_Active,
    VI_First_Fault_Type := GVL_SYSTEM_HEALTH.G_First_Fault_Type,
    VI_First_Fault_Source := GVL_SYSTEM_HEALTH.G_First_Fault_Source
);

// Gateway intent execution
fbSystemGatewayIntent(
    VI_System_Time_MS := GVL_TIME_SERVICE.G_Now_MS,
    VI_IsActivePLC := GVL_STATUS.G_Is_Active_PLC,
    VI_Gateway_Writes_Allowed := NOT GVL_STATUS.G_Diagnostics.Operator_Action_Blocked,
    VIO_FloorHeating_Temps := GVL_STATE.G_Floor_Temps,
    VIO_Zone_Valve_States := GVL_STATE.G_Zone_Valves,
    VIO_Lighting_Base_Levels := GVL_STATE.G_Lighting_Levels,
    VIO_Scenario_Req_Gateway := L_Scenario_Req_Gateway
);

GVL_INTENT_USER.I_Scenario_Request := L_Scenario_Req_Gateway;
          
END_PROGRAM

PROGRAM PRG_Debug_View
  VAR
    L_i : INT;
    L_MaxWeight : REAL;
    L_MinWeight : REAL;
    L_Weight : REAL;
    L_Index : INT;
  END_VAR

            GVL_DEBUG_VIEW.D_Current_Time_MS := GVL_TIME_SERVICE.G_Now_MS;

GVL_DEBUG_VIEW.D_Safety_Mode := GVL_SAFETY_SHUTDOWN.G_Safety_Mode;
GVL_DEBUG_VIEW.D_Safety_Active := (GVL_SAFETY_SHUTDOWN.G_Safety_Mode <> NORMAL);
GVL_DEBUG_VIEW.D_Recovery_Phase := GVL_SAFETY_RECOVERY.G_Recovery_Phase;
GVL_DEBUG_VIEW.D_Recovery_Active := GVL_SAFETY_RECOVERY.G_Recovery_Active;

GVL_DEBUG_VIEW.D_Current_Scenario := GVL_INTENT_BEHAVIOR.I_Selected_Scenario_Text;
GVL_DEBUG_VIEW.D_Behavior_Reason := GVL_INTENT_BEHAVIOR.I_Reason_Text;

GVL_DEBUG_VIEW.D_Score_Night := GVL_INTENT_BEHAVIOR.I_Score_Night;
GVL_DEBUG_VIEW.D_Score_Preheat := GVL_INTENT_BEHAVIOR.I_Score_Preheat;
GVL_DEBUG_VIEW.D_Score_VentBoost := GVL_INTENT_BEHAVIOR.I_Score_Vent_Boost;
GVL_DEBUG_VIEW.D_Score_AccessSecure := GVL_INTENT_BEHAVIOR.I_Score_Access_Secure;

GVL_DEBUG_VIEW.D_Intent_Night := GVL_INTENT_BEHAVIOR.I_Request_Night_Mode;
GVL_DEBUG_VIEW.D_Intent_Comfort := GVL_INTENT_BEHAVIOR.I_Request_Comfort_Mode;
GVL_DEBUG_VIEW.D_Intent_VentBoost := GVL_INTENT_BEHAVIOR.I_Request_Ventilation_Boost;
GVL_DEBUG_VIEW.D_Intent_AccessSecure := GVL_INTENT_BEHAVIOR.I_Request_Access_Secure_Mode;

GVL_DEBUG_VIEW.D_Heating_Block := GVL_COMMAND_SHADOW.G_Heating_Block;
GVL_DEBUG_VIEW.D_Vent_Stop := GVL_COMMAND_SHADOW.G_Vent_Stop;
GVL_DEBUG_VIEW.D_Water_Block := GVL_COMMAND_SHADOW.G_Water_Block;
GVL_DEBUG_VIEW.D_Access_Open_Active := GVL_COMMAND_SHADOW.G_Gate_Open OR GVL_COMMAND_SHADOW.G_Wicket_Open;

GVL_DEBUG_VIEW.D_Global_Reason := GVL_EXPLAINABILITY.G_Last_Global_Reason_Text;
GVL_DEBUG_VIEW.D_Behavior_Why_Active := GVL_EXPLAINABILITY.G_Behavior_Why_Active;
GVL_DEBUG_VIEW.D_Heating_Why_Blocked := GVL_EXPLAINABILITY.G_Heating_Why_Blocked;
GVL_DEBUG_VIEW.D_Vent_Why_Stopped := GVL_EXPLAINABILITY.G_Vent_Why_Stopped;
GVL_DEBUG_VIEW.D_Water_Why_Closed := GVL_EXPLAINABILITY.G_Water_Why_Closed;
GVL_DEBUG_VIEW.D_Access_Why_Opened := GVL_EXPLAINABILITY.G_Access_Why_Opened;

// SENSOR QUALITY → HMI
GVL_DEBUG_VIEW.D_Input_Source_Valid := GVL_INPUT.IN_Source_Valid;
GVL_DEBUG_VIEW.D_Input_Degraded := GVL_INPUT.IN_Input_Degraded;
GVL_DEBUG_VIEW.D_Sensor_Fault := GVL_INPUT.IN_Sensor_Fault;
GVL_DEBUG_VIEW.D_Validation_Failed := GVL_INPUT.IN_Validation_Failed;
GVL_DEBUG_VIEW.D_Anomaly_Detected := GVL_INPUT.IN_Anomaly_Detected;
GVL_DEBUG_VIEW.D_Validation_Reason := GVL_INPUT.IN_Validation_Reason;
GVL_DEBUG_VIEW.D_Anomaly_Reason := GVL_INPUT.IN_Anomaly_Reason;
GVL_DEBUG_VIEW.D_Last_Invalid_Zone := GVL_INPUT.IN_Last_Invalid_Zone;
GVL_DEBUG_VIEW.D_Min_Zone_Confidence := GVL_INPUT.IN_Min_Zone_Confidence;
GVL_DEBUG_VIEW.D_Worst_Zone := GVL_INPUT.IN_Worst_Zone;

GVL_DEBUG_VIEW.D_Adapt_Profile := GVL_BEHAVIOR_ADAPT.G_Adapt_Profile;

IF GVL_BEHAVIOR_ADAPT.G_Adapt_Profile = ADAPT_PROFILE_STABLE THEN
    GVL_DEBUG_VIEW.D_Adapt_Profile_Text := 'STABLE';
ELSIF GVL_BEHAVIOR_ADAPT.G_Adapt_Profile = ADAPT_PROFILE_BALANCED THEN
    GVL_DEBUG_VIEW.D_Adapt_Profile_Text := 'BALANCED';
ELSE
    GVL_DEBUG_VIEW.D_Adapt_Profile_Text := 'AGGRESSIVE';
END_IF;

L_MaxWeight := 0.0;
L_MinWeight := 9999.0;
GVL_DEBUG_VIEW.D_Main_VentBoost_Zone := 0;

FOR L_i := 1 TO GVL_CONSTANTS.C_MAX_ZONES DO
    L_Weight := GVL_BEHAVIOR_ADAPT.G_VentBoost_Zone_Adapt[L_i].Zone_Weight;
    IF L_Weight > L_MaxWeight THEN
        L_MaxWeight := L_Weight;
        GVL_DEBUG_VIEW.D_Main_VentBoost_Zone := L_i;
        GVL_DEBUG_VIEW.D_Main_VentBoost_Zone_Weight := L_Weight;
        GVL_DEBUG_VIEW.D_Main_VentBoost_Zone_Confidence :=
            GVL_BEHAVIOR_ADAPT.G_VentBoost_Zone_Adapt[L_i].Confidence;
    END_IF;
    IF L_Weight < L_MinWeight THEN
        L_MinWeight := L_Weight;
    END_IF;
END_FOR;

GVL_DEBUG_VIEW.D_Max_VentBoost_Zone_Weight := L_MaxWeight;
GVL_DEBUG_VIEW.D_Min_VentBoost_Zone_Weight := L_MinWeight;

L_Index := GVL_TRACE.G_Trace_Write_Index - 1;
IF L_Index < 1 THEN
    L_Index := 200;
END_IF;

GVL_DEBUG_VIEW.D_Last_Trace_Text := GVL_TRACE.G_Trace_Buffer[L_Index].Text;
GVL_DEBUG_VIEW.D_Last_Trace_Time_MS := GVL_TRACE.G_Trace_Buffer[L_Index].Timestamp_MS;
GVL_DEBUG_VIEW.D_Last_Trace_Reason := GVL_TRACE.G_Trace_Buffer[L_Index].Reason_Code;
          
END_PROGRAM

PROGRAM PRG_Authority_Resurrection_Boundary_Governor

            IF GVL_RECOVERY_REACTIVATION_CONTROL_FABRIC.Recovery_Reactivation_Control_Granted
AND NOT GVL_AUTHORITY_RESURRECTION_BOUNDARY_FABRIC.Partial_Recovery_Authority_Leak
AND NOT GVL_AUTHORITY_RESURRECTION_BOUNDARY_FABRIC.Unsafe_Authority_Resurrection_Detected
AND NOT GVL_AUTHORITY_RESURRECTION_BOUNDARY_FABRIC.Resurrection_Authority_Fork_Detected THEN

    GVL_AUTHORITY_RESURRECTION_BOUNDARY_FABRIC.Authority_Resurrection_Boundary_Valid := TRUE;
    GVL_AUTHORITY_RESURRECTION_BOUNDARY_FABRIC.Authority_Resurrection_Bounded := TRUE;
    GVL_AUTHORITY_RESURRECTION_BOUNDARY_FABRIC.Authority_Recovery_Lineage_Stable := TRUE;
    GVL_AUTHORITY_RESURRECTION_BOUNDARY_FABRIC.Distributed_Authority_Recovery_Consensus := TRUE;
END_IF;
          
END_PROGRAM

PROGRAM PRG_System_BlackBox
  VAR
    fbBlackBox : FB_BlackBox_Recorder;
    L_BB_Record : ST_BlackBox_Record;
    L_BB_Freeze : BOOL;
    L_BB_Gas_Active : BOOL;
    L_BB_Fire_Active : BOOL;
    L_BB_Flood_Active : BOOL;
  END_VAR

            // BlackBox must record authoritative safety truth and latches,
// not stale alarm projection fields.
L_BB_Gas_Active := GVL_HEALTH_BRIDGE.G_Gas_Detected OR GVL_HEALTH_BRIDGE.G_CO_Alarm_Level OR GVL_STATE.G_Safety_Gas_Latched;
L_BB_Fire_Active := GVL_HEALTH_BRIDGE.G_Smoke_Detected OR GVL_STATE.G_Safety_Smoke_Latched;
L_BB_Flood_Active := GVL_HEALTH_BRIDGE.G_Leak_Detected OR GVL_STATE.G_Safety_Leak_Latched;

L_BB_Record.Timestamp := GVL_TIME_SERVICE.G_Now_MS;
L_BB_Record.PLC_Active_ID := GVL_STATUS.G_PLC_ID;
L_BB_Record.Gas_Methane_LEL := GVL_STATE.G_Methane_Sensors[1];
L_BB_Record.Gas_CO_PPM := GVL_STATE.G_CO_Sensors[1];
L_BB_Record.Flood_Active := L_BB_Flood_Active;
L_BB_Record.Fire_Active := L_BB_Fire_Active;

L_BB_Record.System_Mode := TO_BYTE(TO_INT(GVL_STATE.G_System_Mode));
L_BB_Record.First_Fault_Type := TO_BYTE(GVL_SYSTEM_HEALTH.G_First_Fault_Type);
L_BB_Record.First_Fault_Source := TO_BYTE(GVL_SYSTEM_HEALTH.G_First_Fault_Source);
L_BB_Record.First_Fault_Active := GVL_SYSTEM_HEALTH.G_First_Fault_Active;
L_BB_Record.System_Severity := TO_BYTE(GVL_SYSTEM_HEALTH.G_System_Severity);
L_BB_Record.Root_Cause := TO_BYTE(GVL_SYSTEM_HEALTH.G_Root_Cause);
L_BB_Record.Watchdog_Fault := GVL_SYSTEM_HEALTH.G_Watchdog_Fault;

L_BB_Freeze := L_BB_Gas_Active OR L_BB_Fire_Active OR L_BB_Flood_Active OR GVL_SYSTEM_HEALTH.G_First_Fault_Active;

fbBlackBox(
    VI_Current_Data := L_BB_Record,
    VI_Freeze := L_BB_Freeze
);
          
END_PROGRAM

PROGRAM PRG_Convergence_Governor
  VAR
    L_Now_MS : UDINT;
    L_Healthy : BOOL := TRUE;
    L_Error_Code : UDINT := 0;
    L_Error_Text : STRING(160) := '';
    L_Recent_Invalidation : BOOL;
    L_Epoch_Advancement_Healthy : BOOL;
  END_VAR

            L_Now_MS := GVL_STATUS.G_System_Time_MS;
L_Healthy := TRUE;
L_Error_Code := 0;
L_Error_Text := '';

GVL_CONVERGENCE.Convergence_Runtime_Barrier_OK :=
    GVL_RUNTIME_EPOCH.Runtime_Runtime_Barrier_OK
    AND GVL_RUNTIME_EPOCH.Runtime_IO_Publication_Allowed;

GVL_CONVERGENCE.Convergence_Runtime_Snapshot_OK :=
    GVL_RUNTIME_SNAPSHOT.Snapshot_Frozen
    AND GVL_RUNTIME_SNAPSHOT.Snapshot_Publication_Allowed
    AND GVL_RUNTIME_SNAPSHOT.Snapshot_Copy_Valid
    AND GVL_RUNTIME_SNAPSHOT.Snapshot_Isolation_Valid
    AND GVL_RUNTIME_SNAPSHOT.Snapshot_Runtime_Authority_Valid
    AND NOT GVL_RUNTIME_SNAPSHOT.Snapshot_Mutation_Detected;

GVL_CONVERGENCE.Convergence_Distributed_Snapshot_OK :=
    GVL_DISTRIBUTED_SNAPSHOT.Distributed_Publication_Reconciled
    AND GVL_DISTRIBUTED_SNAPSHOT.Distributed_Publication_Freeze_Valid
    AND GVL_DISTRIBUTED_SNAPSHOT.Distributed_Snapshot_Consistent;

GVL_CONVERGENCE.Convergence_Distributed_Commit_OK :=
    GVL_DISTRIBUTED_COMMIT.Distributed_Commit_Valid
    AND GVL_DISTRIBUTED_COMMIT.Publication_Prepare_Valid
    AND GVL_DISTRIBUTED_COMMIT.Publication_Commit_Confirmed
    AND NOT GVL_DISTRIBUTED_COMMIT.Peer_Commit_Mismatch
    AND NOT GVL_DISTRIBUTED_COMMIT.Commit_Lease_Expired;

GVL_CONVERGENCE.Convergence_Semantic_Progress_OK :=
    GVL_SEMANTIC_PROGRESS.Semantic_Forward_Progress_Valid
    AND GVL_SEMANTIC_PROGRESS.Semantic_Execution_Continuity_OK
    AND NOT GVL_SEMANTIC_PROGRESS.Semantic_Stagnation_Detected
    AND NOT GVL_SEMANTIC_PROGRESS.Semantic_Replay_Suspected
    AND NOT GVL_SEMANTIC_PROGRESS.Semantic_Livelock_Suspected
    AND NOT GVL_SEMANTIC_PROGRESS.Semantic_Deadlock_Suspected
    AND NOT GVL_SEMANTIC_PROGRESS.Semantic_Progress_Lease_Expired
    AND NOT GVL_SEMANTIC_PROGRESS.Semantic_Progress_Quarantine_Active;

GVL_CONVERGENCE.Convergence_Output_Freshness_OK :=
    GVL_RUNTIME_EPOCH.Runtime_Runtime_Barrier_OK
    AND GVL_RUNTIME_EPOCH.Runtime_IO_Publication_Allowed
    AND GVL_RUNTIME_SNAPSHOT.Snapshot_Frozen
    AND GVL_RUNTIME_SNAPSHOT.Snapshot_Publication_Allowed
    AND GVL_RUNTIME_SNAPSHOT.Snapshot_Copy_Valid
    AND GVL_RUNTIME_SNAPSHOT.Snapshot_Isolation_Valid
    AND NOT GVL_RUNTIME_SNAPSHOT.Snapshot_Mutation_Detected
    AND GVL_DISTRIBUTED_SNAPSHOT.Distributed_Publication_Reconciled
    AND GVL_DISTRIBUTED_SNAPSHOT.Distributed_Publication_Freeze_Valid
    AND GVL_DISTRIBUTED_SNAPSHOT.Distributed_Snapshot_Consistent
    AND GVL_DISTRIBUTED_COMMIT.Distributed_Commit_Valid
    AND GVL_DISTRIBUTED_COMMIT.Publication_Prepare_Valid
    AND GVL_DISTRIBUTED_COMMIT.Publication_Commit_Confirmed
    AND NOT GVL_DISTRIBUTED_COMMIT.Peer_Commit_Mismatch
    AND NOT GVL_DISTRIBUTED_COMMIT.Commit_Lease_Expired
    AND GVL_OUTPUT_EPOCH.Output_Publication_Valid
    AND GVL_OUTPUT_EPOCH.Output_Runtime_Epoch_Valid
    AND NOT GVL_OUTPUT_EPOCH.Output_Lease_Expired
    AND NOT GVL_OUTPUT_EPOCH.Output_Forced_Safe_Decay
    AND GVL_COMMAND_VERIFY.PreOutput_Barrier_OK
    AND NOT GVL_COMMAND_VERIFY.PreOutput_Block_IO;

// Epoch advancement freshness.
L_Epoch_Advancement_Healthy :=
    (GVL_SEMANTIC_PROGRESS.Semantic_Runtime_Barrier_Epoch -
     GVL_SEMANTIC_PROGRESS.Semantic_Last_Runtime_Barrier_Epoch) <= 2
    AND
    (GVL_SEMANTIC_PROGRESS.Semantic_Distributed_Commit_Epoch -
     GVL_SEMANTIC_PROGRESS.Semantic_Last_Distributed_Commit_Epoch) <= 2
    AND
    (GVL_SEMANTIC_PROGRESS.Semantic_Output_Publication_Epoch -
     GVL_SEMANTIC_PROGRESS.Semantic_Last_Output_Publication_Epoch) <= 2;

// Oscillation damping window.
L_Recent_Invalidation :=
    (L_Now_MS - GVL_CONVERGENCE.Convergence_Last_Invalidation_MS) < 30000;

IF NOT GVL_CONVERGENCE.Convergence_Runtime_Barrier_OK THEN
    L_Healthy := FALSE;
    L_Error_Code := 18000;
    L_Error_Text := 'Runtime barrier convergence invalid';
END_IF;

IF L_Healthy AND NOT GVL_CONVERGENCE.Convergence_Runtime_Snapshot_OK THEN
    L_Healthy := FALSE;
    L_Error_Code := 18001;
    L_Error_Text := 'Runtime snapshot convergence invalid';
END_IF;

IF L_Healthy AND NOT GVL_CONVERGENCE.Convergence_Distributed_Snapshot_OK THEN
    L_Healthy := FALSE;
    L_Error_Code := 18002;
    L_Error_Text := 'Distributed snapshot convergence invalid';
END_IF;

IF L_Healthy AND NOT GVL_CONVERGENCE.Convergence_Distributed_Commit_OK THEN
    L_Healthy := FALSE;
    L_Error_Code := 18003;
    L_Error_Text := 'Distributed commit convergence invalid';
END_IF;

IF L_Healthy AND NOT GVL_CONVERGENCE.Convergence_Semantic_Progress_OK THEN
    L_Healthy := FALSE;
    L_Error_Code := 18004;
    L_Error_Text := 'Semantic progress convergence invalid';
END_IF;

IF L_Healthy AND NOT GVL_CONVERGENCE.Convergence_Output_Freshness_OK THEN
    L_Healthy := FALSE;
    L_Error_Code := 18005;
    L_Error_Text := 'Output freshness convergence invalid';
END_IF;

IF L_Healthy AND NOT L_Epoch_Advancement_Healthy THEN
    L_Healthy := FALSE;
    L_Error_Code := 18006;
    L_Error_Text := 'Epoch advancement freshness invalid';
END_IF;

IF L_Healthy AND L_Recent_Invalidation THEN
    L_Healthy := FALSE;
    L_Error_Code := 18007;
    L_Error_Text := 'Convergence oscillation damping active';
END_IF;

IF L_Healthy THEN
    GVL_CONVERGENCE.Convergence_Healthy_Observed := TRUE;

    GVL_CONVERGENCE.Recovery_Stable_Cycle_Count :=
        GVL_CONVERGENCE.Recovery_Stable_Cycle_Count + 1;

    IF GVL_CONVERGENCE.Convergence_Last_Healthy_MS = 0 THEN
        GVL_CONVERGENCE.Convergence_Last_Healthy_MS := L_Now_MS;
    END_IF;

    GVL_CONVERGENCE.Recovery_Stable_Time_MS :=
        L_Now_MS - GVL_CONVERGENCE.Convergence_Last_Healthy_MS;

    IF (GVL_CONVERGENCE.Recovery_Stable_Cycle_Count >= GVL_CONVERGENCE.Convergence_Min_Stable_Cycles)
    AND (GVL_CONVERGENCE.Recovery_Stable_Time_MS >= GVL_CONVERGENCE.Convergence_Min_Stable_Time_MS)
    THEN
        GVL_CONVERGENCE.Convergence_Lease_OK := TRUE;
        GVL_CONVERGENCE.Convergence_Release_Allowed := TRUE;
    ELSE
        GVL_CONVERGENCE.Convergence_Lease_OK := FALSE;
        GVL_CONVERGENCE.Convergence_Release_Allowed := FALSE;
    END_IF;

    GVL_CONVERGENCE.Convergence_Last_Error_Code := 0;
    GVL_CONVERGENCE.Convergence_Last_Error_Text := '';
ELSE
    GVL_CONVERGENCE.Convergence_Healthy_Observed := FALSE;

    GVL_CONVERGENCE.Recovery_Stable_Cycle_Count := 0;
    GVL_CONVERGENCE.Recovery_Stable_Time_MS := 0;

    GVL_CONVERGENCE.Convergence_Lease_OK := FALSE;
    GVL_CONVERGENCE.Convergence_Release_Allowed := FALSE;

    GVL_CONVERGENCE.Convergence_Last_Healthy_MS := 0;
    GVL_CONVERGENCE.Convergence_Last_Invalidation_MS := L_Now_MS;

    GVL_CONVERGENCE.Convergence_Invalidation_Count :=
        GVL_CONVERGENCE.Convergence_Invalidation_Count + 1;

    // Oscillation quarantine.
    IF GVL_CONVERGENCE.Convergence_Invalidation_Count > 5 THEN
        GVL_CONVERGENCE.Convergence_Oscillation_Quarantine_Active := TRUE;
    END_IF;

    GVL_CONVERGENCE.Convergence_Last_Error_Code := L_Error_Code;
    GVL_CONVERGENCE.Convergence_Last_Error_Text := L_Error_Text;
END_IF;
          
END_PROGRAM

PROGRAM PRG_Control_Temporal_Coherence_Governor
  VAR
    L_Now_MS : UDINT;
    L_Control_Valid : BOOL := TRUE;
    L_Error_Code : UDINT := 0;
    L_Error_Text : STRING(160) := '';
  END_VAR

            L_Now_MS := GVL_STATUS.G_System_Time_MS;
L_Control_Valid := TRUE;
L_Error_Code := 0;
L_Error_Text := '';

// Fail-safe defaults.
GVL_CONTROL_TIMING_FABRIC.Control_Temporal_Coherence_Valid := FALSE;
GVL_CONTROL_TIMING_FABRIC.Control_Temporal_Coherence_Granted := FALSE;
GVL_CONTROL_TIMING_FABRIC.Control_Temporal_Coherence_Quarantine_Active := TRUE;

GVL_CONTROL_TIMING_FABRIC.Loop_Sampling_Coherent := FALSE;
GVL_CONTROL_TIMING_FABRIC.Feedback_Freshness_Valid := FALSE;
GVL_CONTROL_TIMING_FABRIC.PID_Phase_Alignment_Valid := FALSE;
GVL_CONTROL_TIMING_FABRIC.Cross_Loop_Temporal_Stable := FALSE;
GVL_CONTROL_TIMING_FABRIC.Multi_Rate_Causality_Coherent := FALSE;

// Global authority synchronization required.
IF NOT GVL_GLOBAL_AUTHORITY_SYNC.Global_Authority_Sync_Granted THEN
    L_Control_Valid := FALSE;
    L_Error_Code := 35000;
    L_Error_Text := 'Global authority synchronization not granted';
END_IF;

// Temporal aliasing detectors.
IF GVL_CONTROL_TIMING_FABRIC.PID_Phase_Skew_Detected THEN
    L_Control_Valid := FALSE;
    L_Error_Code := 35001;
    L_Error_Text := 'PID phase skew detected';
END_IF;

IF GVL_CONTROL_TIMING_FABRIC.Sampling_Window_Divergence_Detected THEN
    L_Control_Valid := FALSE;
    L_Error_Code := 35002;
    L_Error_Text := 'Sampling window divergence detected';
END_IF;

IF GVL_CONTROL_TIMING_FABRIC.Feedback_Freshness_Aliasing_Detected THEN
    L_Control_Valid := FALSE;
    L_Error_Code := 35003;
    L_Error_Text := 'Feedback freshness aliasing detected';
END_IF;

IF GVL_CONTROL_TIMING_FABRIC.Cross_Loop_Stabilization_Lag_Detected THEN
    L_Control_Valid := FALSE;
    L_Error_Code := 35004;
    L_Error_Text := 'Cross-loop stabilization lag detected';
END_IF;

IF GVL_CONTROL_TIMING_FABRIC.Multi_Rate_Oscillation_Risk_Detected THEN
    L_Control_Valid := FALSE;
    L_Error_Code := 35005;
    L_Error_Text := 'Multi-rate oscillation risk detected';
END_IF;

IF GVL_CONTROL_TIMING_FABRIC.Distributed_Control_Ringing_Detected THEN
    L_Control_Valid := FALSE;
    L_Error_Code := 35006;
    L_Error_Text := 'Distributed control ringing detected';
END_IF;

// Deterministic control timing validation.
IF L_Control_Valid
AND NOT GVL_CONTROL_TIMING_FABRIC.Control_Snapshot_Epoch_Coherent THEN
    L_Control_Valid := FALSE;
    L_Error_Code := 35010;
    L_Error_Text := 'Control snapshot epoch coherence invalid';
END_IF;

IF L_Control_Valid
AND NOT GVL_CONTROL_TIMING_FABRIC.Feedback_Window_Stable THEN
    L_Control_Valid := FALSE;
    L_Error_Code := 35011;
    L_Error_Text := 'Feedback window unstable';
END_IF;

IF L_Control_Valid
AND NOT GVL_CONTROL_TIMING_FABRIC.Loop_Execution_Phase_Stable THEN
    L_Control_Valid := FALSE;
    L_Error_Code := 35012;
    L_Error_Text := 'Loop execution phase unstable';
END_IF;

IF L_Control_Valid
AND NOT GVL_CONTROL_TIMING_FABRIC.Temporal_Observation_Aligned THEN
    L_Control_Valid := FALSE;
    L_Error_Code := 35013;
    L_Error_Text := 'Temporal observation alignment invalid';
END_IF;

IF L_Control_Valid THEN
    GVL_CONTROL_TIMING_FABRIC.Control_Temporal_Coherence_Valid := TRUE;
    GVL_CONTROL_TIMING_FABRIC.Control_Temporal_Coherence_Granted := TRUE;
    GVL_CONTROL_TIMING_FABRIC.Control_Temporal_Coherence_Quarantine_Active := FALSE;

    GVL_CONTROL_TIMING_FABRIC.Loop_Sampling_Coherent := TRUE;
    GVL_CONTROL_TIMING_FABRIC.Feedback_Freshness_Valid := TRUE;
    GVL_CONTROL_TIMING_FABRIC.PID_Phase_Alignment_Valid := TRUE;
    GVL_CONTROL_TIMING_FABRIC.Cross_Loop_Temporal_Stable := TRUE;
    GVL_CONTROL_TIMING_FABRIC.Multi_Rate_Causality_Coherent := TRUE;

    GVL_CONTROL_TIMING_FABRIC.Control_Timing_Epoch :=
        GVL_GLOBAL_AUTHORITY_SYNC.Global_Authority_Epoch;

    GVL_CONTROL_TIMING_FABRIC.Control_Timing_Epoch_Coherent := TRUE;

    GVL_CONTROL_TIMING_FABRIC.Control_Timing_Last_Update_MS := L_Now_MS;
    GVL_CONTROL_TIMING_FABRIC.Control_Timing_Lease_Expired := FALSE;

    GVL_CONTROL_TIMING_FABRIC.Control_Timing_Last_Error_Code := 0;
    GVL_CONTROL_TIMING_FABRIC.Control_Timing_Last_Error_Text := '';
ELSE
    GVL_CONTROL_TIMING_FABRIC.Control_Temporal_Coherence_Valid := FALSE;
    GVL_CONTROL_TIMING_FABRIC.Control_Temporal_Coherence_Granted := FALSE;
    GVL_CONTROL_TIMING_FABRIC.Control_Temporal_Coherence_Quarantine_Active := TRUE;

    GVL_CONTROL_TIMING_FABRIC.Control_Timing_Lease_Expired := TRUE;

    GVL_CONTROL_TIMING_FABRIC.Control_Timing_Last_Error_Code :=
        L_Error_Code;

    GVL_CONTROL_TIMING_FABRIC.Control_Timing_Last_Error_Text :=
        L_Error_Text;

    GVL_CONTROL_TIMING_FABRIC.Control_Timing_Invalidation_Count :=
        GVL_CONTROL_TIMING_FABRIC.Control_Timing_Invalidation_Count + 1;
END_IF;
          
END_PROGRAM

PROGRAM PRG_Heating
  VAR
    fbHeatingManager : FB_Heating_System_Manager;
    fbDHWManager : FB_DHW_Manager;
    fbDiagnosticsPhase : FB_Heating_Runtime_Diagnostics_Phase;
    fbObserverPhase : FB_Heating_Runtime_Observer_Phase;
    fbMetaSupervisionPublisher : FB_Heating_Runtime_Meta_Supervision_Publisher;
    fbExplainabilityPublisher : FB_Heating_Runtime_Explainability_Publisher;
    fbServiceGatingPhase : FB_Heating_Runtime_Service_Gating_Phase;
    fbStatePublicationPhase : FB_Heating_Runtime_State_Publication_Phase;
    fbOutputProjectionPhase : FB_Heating_Runtime_Output_Projection_Phase;
    L_Runtime_Context : ST_Heating_Runtime_Context;
    L_i : INT;
    L_Current_Hour : UINT;
    L_Boiler_Modulation_REAL : ARRAY[1..GVL_CONSTANTS.C_MAX_BOILERS] OF REAL;
    L_Room_Temps_Normalized : ARRAY[1..GVL_CONSTANTS.C_MAX_ZONES] OF REAL;
    L_Floor_Temps_Normalized : ARRAY[1..GVL_CONSTANTS.C_MAX_HEATING_CIRCUITS] OF REAL;
    L_Outdoor_Temp_Normalized : REAL;
    L_Heating_Emergency_Stop : BOOL;
    L_Heating_Gas_Safety_Stop : BOOL;
    L_Distributed_Execute_Allowed : BOOL;
    L_Distributed_Orchestrate_Allowed : BOOL;
    L_Distributed_Projection_Allowed : BOOL;
    L_Zone_Valves : ARRAY[1..GVL_CONSTANTS.C_MAX_HEATING_CIRCUITS] OF BOOL;
    L_Manifold_Pumps : ARRAY[1..GVL_CONSTANTS.C_MAX_MANIFOLDS] OF BOOL;
    L_Manifold_Valves : ARRAY[1..GVL_CONSTANTS.C_MAX_MANIFOLDS] OF REAL;
    L_Boiler_OT_Enable : ARRAY[1..GVL_CONSTANTS.C_MAX_BOILERS] OF BOOL;
    L_Boiler_OT_Setpoint : ARRAY[1..GVL_CONSTANTS.C_MAX_BOILERS] OF REAL;
    L_Backup_Circulation_Pump : BOOL;
    L_Electric_Heater_Enable : BOOL;
    L_Freeze_Risk_Status : BOOL;
    L_Manifold_Status : ARRAY[1..GVL_CONSTANTS.C_MAX_MANIFOLDS] OF ST_Manifold_Status;
    L_Boiler_Status : ARRAY[1..GVL_CONSTANTS.C_MAX_BOILERS] OF ST_Boiler_Status;
    L_DHW_Heating_Pump : BOOL;
    L_DHW_Circ_Pump : BOOL;
    L_DHW_Status : ST_DHW_Status;
  END_VAR

            FOR L_i := 1 TO GVL_CONSTANTS.C_MAX_BOILERS DO
    L_Boiler_Modulation_REAL[L_i] := TO_REAL(GVL_IO.AI_Boiler_Modulation[L_i]);
END_FOR;

L_Current_Hour := TO_UINT(GVL_TIME_SERVICE.G_Time_Of_Day_MS / 3600000);

L_Outdoor_Temp_Normalized := GVL_INPUT.IN_Outdoor_Temp;

FOR L_i := 1 TO GVL_CONSTANTS.C_MAX_ZONES DO
    L_Room_Temps_Normalized[L_i] := GVL_INPUT.IN_Room_Temps[L_i];
END_FOR;

FOR L_i := 1 TO GVL_CONSTANTS.C_MAX_HEATING_CIRCUITS DO
    L_Floor_Temps_Normalized[L_i] := GVL_INPUT.IN_Floor_Temps[L_i];
END_FOR;

L_Heating_Emergency_Stop := GVL_COMMAND_SHADOW.G_Heating_Emergency_Stop;
L_Heating_Gas_Safety_Stop := GVL_COMMAND_SHADOW.G_Heating_Gas_Safety_Stop OR GVL_STATE.G_Safety_Gas_Latched;

// Centralized distributed runtime governance.
// Freeze protection and gas safety semantics remain authoritative.
L_Distributed_Execute_Allowed :=
    GVL_Distributed_Execution_Gates.G_Can_Execute;

L_Distributed_Orchestrate_Allowed :=
    GVL_Distributed_Execution_Gates.G_Can_Orchestrate;

L_Distributed_Projection_Allowed :=
    GVL_Distributed_Execution_Gates.G_Can_Own_Projection;

L_Runtime_Context.Runtime_Enabled := TRUE;
L_Runtime_Context.Runtime_Ready := TRUE;
L_Runtime_Context.Runtime_Fault := FALSE;
L_Runtime_Context.Current_Phase := E_Heating_Runtime_Phase.HRP_IDLE;

L_Runtime_Context.Allow_DHW_Phase :=
    L_Distributed_Execute_Allowed;

L_Runtime_Context.Allow_Heating_Phase :=
    L_Distributed_Orchestrate_Allowed;

L_Runtime_Context.Allow_Service_Gating_Phase := TRUE;
L_Runtime_Context.Allow_State_Publication_Phase := TRUE;
L_Runtime_Context.Allow_Diagnostics_Phase := TRUE;

L_Runtime_Context.Allow_Output_Projection_Phase :=
    L_Distributed_Projection_Allowed;

L_Runtime_Context.DHW_Executed := FALSE;
L_Runtime_Context.Heating_Executed := FALSE;
L_Runtime_Context.Service_Gating_Executed := FALSE;
L_Runtime_Context.State_Publication_Executed := FALSE;
L_Runtime_Context.Diagnostics_Executed := FALSE;
L_Runtime_Context.Output_Projection_Executed := FALSE;

L_Runtime_Context.DHW_Before_Heating_Valid := TRUE;
L_Runtime_Context.State_Publication_Before_Diagnostics_Valid := TRUE;
L_Runtime_Context.Output_Projection_Last_Valid := TRUE;

L_Runtime_Context.Diagnostics_Isolation_Valid := TRUE;
L_Runtime_Context.Explainability_Isolation_Valid := TRUE;
L_Runtime_Context.Safety_Isolation_Valid := TRUE;
L_Runtime_Context.OpenTherm_Ownership_Valid := TRUE;
L_Runtime_Context.Cascade_Ownership_Valid := TRUE;

IF NOT L_Distributed_Execute_Allowed THEN
    L_Runtime_Context.Runtime_Status_Code := 20;
    L_Runtime_Context.Runtime_Status_Text :=
        'Heating runtime blocked by distributed governance';
ELSE
    L_Runtime_Context.Runtime_Status_Code := 1;
    L_Runtime_Context.Runtime_Status_Text :=
        'Heating runtime nominal';
END_IF;

L_Runtime_Context.Current_Phase := E_Heating_Runtime_Phase.HRP_IDLE;

fbObserverPhase(
    VI_Authorization_Stage := TRUE,
    VI_Finalization_Stage := FALSE,
    VI_Runtime_Context := L_Runtime_Context,
    VI_Diagnostics_Valid := TRUE
);

IF L_Distributed_Execute_Allowed THEN

    L_Runtime_Context.Current_Phase := E_Heating_Runtime_Phase.HRP_DHW;

    fbDHWManager(
        VI_System_Time_MS := GVL_STATUS.G_System_Time_MS,
        VI_Current_TOD := GVL_STATUS.G_Current_TOD,
        VI_IsActivePLC := GVL_STATUS.G_Is_Active_PLC,
        VI_Temp := GVL_STATE.G_DHW_Temp,
        VI_Pressure := GVL_STATE.G_DHW_Pressure,
        VI_Config := GVL_CONFIG.G_DHW_Config,
        VI_Current_Day_Of_Week := GVL_STATUS.G_Current_Day,
        VI_IO_Modules_Online := GVL_STATUS.G_IO_Modules_Online,
        VI_Reset_Errors := GVL_INTENT_USER.I_Reset_Errors,
        VI_Emergency_Stop := L_Heating_Emergency_Stop,
        VI_System_Mode := GVL_STATE.G_System_Mode,
        VO_Status => L_DHW_Status,
        VO_Heating_Pump => L_DHW_Heating_Pump,
        VO_Circ_Pump => L_DHW_Circ_Pump
    );

    L_Runtime_Context.DHW_Executed := TRUE;

END_IF;

IF L_Heating_Gas_Safety_Stop THEN
    L_DHW_Heating_Pump := FALSE;
    L_DHW_Status.Heating_Pump_On := FALSE;
END_IF;

IF L_Distributed_Orchestrate_Allowed THEN

    L_Runtime_Context.Current_Phase := E_Heating_Runtime_Phase.HRP_HEATING;

    fbHeatingManager(
        VI_System_Mode := GVL_STATE.G_System_Mode,
        VI_System_Time_MS := GVL_STATUS.G_System_Time_MS,
        VI_IsActivePLC := GVL_STATUS.G_Is_Active_PLC,
        VI_Outdoor_Temp := L_Outdoor_Temp_Normalized,
        VI_Config := GVL_CONFIG.G_Heating_Config,
        VI_Tariff := GVL_CONFIG.G_HMI_Tariff_Settings,
        VI_Current_Hour := L_Current_Hour,
        VI_DHW_Heating_Demand := L_DHW_Heating_Pump,
        VI_DHW_Target_Temp := GVL_CONFIG.G_DHW_Config.Target_Temp,
        VI_Emergency_Stop := L_Heating_Emergency_Stop,
        VI_Gas_Safety_Stop := L_Heating_Gas_Safety_Stop,
        VI_Boiler_Error_Status := GVL_STATE.G_Boiler_Error,
        VI_Boiler_OT_Online := GVL_STATE.G_Boiler_OT_Online,
        VI_Boiler_Modulation := L_Boiler_Modulation_REAL,
        VI_Floor_Temps := L_Floor_Temps_Normalized,
        VI_Room_Temps := L_Room_Temps_Normalized,
        VI_Manifold_Pressures := GVL_STATE.G_Manifold_Pressures,
        VI_Manifold_Currents := GVL_STATE.G_Manifold_Currents,
        VI_Manifold_Temps_Supply := GVL_STATE.G_Manifold_T_Supply,
        VI_Manifold_Temps_Return := GVL_STATE.G_Manifold_T_Return,
        VI_Boiler_Flame_Status := GVL_STATE.G_Boiler_Flame,
        VI_Zone_Configs := GVL_CONFIG.G_HMI_FloorHeating_Configs,
        VI_Rule_Actions := GVL_STATE.G_Rule_Actions,
        VI_IO_Modules_Online := GVL_STATUS.G_IO_Modules_Online,
        VI_Manifold_End_Switches := GVL_STATE.G_Manifold_End_Switches,
        VI_Valve_Test_Config := GVL_CONFIG.G_Valve_Test_Config,
        VO_Manifold_Valves => L_Manifold_Valves,
        VO_Manifold_Pumps => L_Manifold_Pumps,
        VO_Zone_Valves => L_Zone_Valves,
        VO_Boiler_OT_Enable => L_Boiler_OT_Enable,
        VO_Boiler_OT_Setpoint => L_Boiler_OT_Setpoint,
        VO_Backup_Circulation_Pump => L_Backup_Circulation_Pump,
        VO_Electric_Heater_Enable => L_Electric_Heater_Enable,
        VO_Freeze_Risk_Status => L_Freeze_Risk_Status,
        VO_Status => L_Manifold_Status,
        VO_Boiler_Status => L_Boiler_Status
    );

    L_Runtime_Context.Heating_Executed := TRUE;

END_IF;

L_Runtime_Context.Current_Phase := E_Heating_Runtime_Phase.HRP_SERVICE_GATING;

fbServiceGatingPhase(
    VI_Enable := TRUE,
    VIO_Manifold_Pumps := L_Manifold_Pumps,
    VIO_Backup_Circulation_Pump := L_Backup_Circulation_Pump,
    VIO_Electric_Heater_Enable := L_Electric_Heater_Enable,
    VIO_DHW_Heating_Pump := L_DHW_Heating_Pump,
    VIO_DHW_Circ_Pump := L_DHW_Circ_Pump,
    VIO_DHW_Status := L_DHW_Status,
    VIO_Freeze_Risk_Status := L_Freeze_Risk_Status
);

L_Runtime_Context.Service_Gating_Executed := fbServiceGatingPhase.VO_Executed;
L_Runtime_Context.Safety_Isolation_Valid := fbServiceGatingPhase.VO_Valid;

L_Runtime_Context.Current_Phase := E_Heating_Runtime_Phase.HRP_STATE_PUBLICATION;

fbStatePublicationPhase(
    VI_Enable := TRUE,
    VI_Zone_Valves := L_Zone_Valves,
    VI_Manifold_Pumps := L_Manifold_Pumps,
    VI_Manifold_Valves := L_Manifold_Valves,
    VI_Boiler_OT_Enable := L_Boiler_OT_Enable,
    VI_Boiler_OT_Setpoint := L_Boiler_OT_Setpoint,
    VI_Backup_Circulation_Pump := L_Backup_Circulation_Pump,
    VI_Electric_Heater_Enable := L_Electric_Heater_Enable,
    VI_Freeze_Risk_Status := L_Freeze_Risk_Status,
    VI_Manifold_Status := L_Manifold_Status,
    VI_Boiler_Status := L_Boiler_Status,
    VI_DHW_Heating_Pump := L_DHW_Heating_Pump,
    VI_DHW_Circ_Pump := L_DHW_Circ_Pump,
    VI_DHW_Status := L_DHW_Status
);

L_Runtime_Context.State_Publication_Executed := fbStatePublicationPhase.VO_Executed;
L_Runtime_Context.State_Publication_Before_Diagnostics_Valid := fbStatePublicationPhase.VO_Valid;

L_Runtime_Context.Current_Phase := E_Heating_Runtime_Phase.HRP_DIAGNOSTICS;

fbDiagnosticsPhase(
    VI_Enable := TRUE,
    VI_System_Time_MS := GVL_STATUS.G_System_Time_MS
);

L_Runtime_Context.Diagnostics_Executed := fbDiagnosticsPhase.VO_Executed;
L_Runtime_Context.Diagnostics_Isolation_Valid := fbDiagnosticsPhase.VO_Valid;

fbObserverPhase(
    VI_Authorization_Stage := FALSE,
    VI_Finalization_Stage := TRUE,
    VI_Runtime_Context := L_Runtime_Context,
    VI_Diagnostics_Valid := L_Runtime_Context.Diagnostics_Isolation_Valid
);

fbMetaSupervisionPublisher(
    VI_Enable := TRUE,
    VI_Runtime_Observation_Valid := GVL_Heating_Runtime_Observation.G_Runtime_Observation_Valid,
    VI_Runtime_Observer_Ready := GVL_Heating_Runtime_Observation.G_Runtime_Observer_Ready,
    VI_Runtime_Observer_Fault := GVL_Heating_Runtime_Observation.G_Runtime_Observer_Fault,
    VI_Runtime_Status_Code := GVL_Heating_Runtime_Observation.G_Runtime_Observation_Status_Code,
    VI_Runtime_Status_Text := GVL_Heating_Runtime_Observation.G_Runtime_Observation_Status_Text
);

GVL_Heating_Runtime_Meta.G_Runtime_Meta_Supervision :=
    fbMetaSupervisionPublisher.VO_Meta;

GVL_Heating_Runtime_Meta.G_Runtime_Meta_Publication_Valid :=
    fbMetaSupervisionPublisher.VO_Publication_Valid;

GVL_Heating_Runtime_Meta.G_Runtime_Meta_Status_Code :=
    fbMetaSupervisionPublisher.VO_Meta.Status_Code;

GVL_Heating_Runtime_Meta.G_Runtime_Meta_Status_Text :=
    fbMetaSupervisionPublisher.VO_Meta.Status_Text;

fbExplainabilityPublisher(
    VI_Enable := TRUE,
    VI_System_Time_MS := GVL_STATUS.G_System_Time_MS,
    VI_Runtime_Context := L_Runtime_Context,
    VI_Runtime_Observation_Valid := GVL_Heating_Runtime_Observation.G_Runtime_Observation_Valid,
    VI_Runtime_Observer_Fault := GVL_Heating_Runtime_Observation.G_Runtime_Observer_Fault,
    VI_Runtime_Status_Code := GVL_Heating_Runtime_Observation.G_Runtime_Observation_Status_Code,
    VI_Runtime_Status_Text := GVL_Heating_Runtime_Observation.G_Runtime_Observation_Status_Text
);

GVL_Heating_Runtime_Explainability.G_Runtime_Phase_Event :=
    fbExplainabilityPublisher.VO_Phase_Event;

GVL_Heating_Runtime_Explainability.G_Runtime_Anomaly :=
    fbExplainabilityPublisher.VO_Anomaly;

GVL_Heating_Runtime_Explainability.G_Runtime_Blackbox_Event :=
    fbExplainabilityPublisher.VO_Blackbox_Event;

GVL_Heating_Runtime_Explainability.G_Runtime_Blackbox_Timeline :=
    fbExplainabilityPublisher.VO_Blackbox_Timeline;

GVL_Heating_Runtime_Explainability.G_Runtime_Event_Buffer :=
    fbExplainabilityPublisher.VO_Event_Buffer;

GVL_Heating_Runtime_Explainability.G_Runtime_Adaptive_Intelligence :=
    fbExplainabilityPublisher.VO_Adaptive_Intelligence;

GVL_Heating_Runtime_Explainability.G_Runtime_Causality_Graph :=
    fbExplainabilityPublisher.VO_Causality_Graph;

GVL_Heating_Runtime_Explainability.G_Runtime_Explainability_Publication_Valid :=
    fbExplainabilityPublisher.VO_Publication_Valid;

GVL_Heating_Runtime_Explainability.G_Runtime_Explainability_Status_Code :=
    fbExplainabilityPublisher.VO_Phase_Event.Status_Code;

GVL_Heating_Runtime_Explainability.G_Runtime_Explainability_Status_Text :=
    fbExplainabilityPublisher.VO_Phase_Event.Status_Text;

IF L_Distributed_Projection_Allowed THEN

    L_Runtime_Context.Current_Phase := E_Heating_Runtime_Phase.HRP_OUTPUT_PROJECTION;

    fbOutputProjectionPhase(
        VI_Enable := TRUE,
        VI_Zone_Valves := L_Zone_Valves,
        VI_Manifold_Pumps := L_Manifold_Pumps,
        VI_Manifold_Valves := L_Manifold_Valves,
        VI_DHW_Heating_Pump := L_DHW_Heating_Pump,
        VI_DHW_Circ_Pump := L_DHW_Circ_Pump,
        VI_Backup_Circulation_Pump := L_Backup_Circulation_Pump,
        VI_Electric_Heater_Enable := L_Electric_Heater_Enable
    );

    L_Runtime_Context.Output_Projection_Executed :=
        fbOutputProjectionPhase.VO_Executed;

    L_Runtime_Context.Output_Projection_Last_Valid :=
        fbOutputProjectionPhase.VO_Valid;

END_IF;

L_Runtime_Context.Current_Phase := E_Heating_Runtime_Phase.HRP_COMPLETE;

// >>> BULK_SYNC_ANCHOR: PRG_Heating <<<
          
END_PROGRAM

PROGRAM PRG_Semantic_Continuity_Authority_Governor
  VAR
    L_Now_MS : UDINT;
    L_Semantic_Valid : BOOL := TRUE;
    L_Error_Code : UDINT := 0;
    L_Error_Text : STRING(160) := '';
  END_VAR

            L_Now_MS := GVL_STATUS.G_System_Time_MS;
L_Semantic_Valid := TRUE;
L_Error_Code := 0;
L_Error_Text := '';

// Fail-safe defaults.
GVL_SEMANTIC_CONTINUITY.Semantic_Continuity_Valid := FALSE;
GVL_SEMANTIC_CONTINUITY.Semantic_Continuity_Granted := FALSE;
GVL_SEMANTIC_CONTINUITY.Semantic_Continuity_Quarantine_Active := TRUE;

GVL_SEMANTIC_CONTINUITY.Operator_Intent_Coherent := FALSE;
GVL_SEMANTIC_CONTINUITY.Policy_Intent_Coherent := FALSE;
GVL_SEMANTIC_CONTINUITY.Adaptive_Behavior_Coherent := FALSE;
GVL_SEMANTIC_CONTINUITY.Recovery_Intent_Coherent := FALSE;
GVL_SEMANTIC_CONTINUITY.Distributed_Semantic_Coherent := FALSE;

// Runtime resource authority required.
IF NOT GVL_RUNTIME_RESOURCE_AUTHORITY.Runtime_Resource_Authority_Granted THEN
    L_Semantic_Valid := FALSE;
    L_Error_Code := 31000;
    L_Error_Text := 'Runtime resource authority not granted';
END_IF;

// Semantic drift detectors.
IF GVL_SEMANTIC_CONTINUITY.Goal_Drift_Detected THEN
    L_Semantic_Valid := FALSE;
    L_Error_Code := 31001;
    L_Error_Text := 'Goal drift detected';
END_IF;

IF GVL_SEMANTIC_CONTINUITY.Policy_Divergence_Detected THEN
    L_Semantic_Valid := FALSE;
    L_Error_Code := 31002;
    L_Error_Text := 'Policy divergence detected';
END_IF;

IF GVL_SEMANTIC_CONTINUITY.Adaptive_Learning_Semantic_Skew THEN
    L_Semantic_Valid := FALSE;
    L_Error_Code := 31003;
    L_Error_Text := 'Adaptive semantic skew detected';
END_IF;

IF GVL_SEMANTIC_CONTINUITY.Recovery_Intent_Mismatch_Detected THEN
    L_Semantic_Valid := FALSE;
    L_Error_Code := 31004;
    L_Error_Text := 'Recovery intent mismatch detected';
END_IF;

IF GVL_SEMANTIC_CONTINUITY.Optimization_Authority_Corruption_Detected THEN
    L_Semantic_Valid := FALSE;
    L_Error_Code := 31005;
    L_Error_Text := 'Optimization authority corruption detected';
END_IF;

IF GVL_SEMANTIC_CONTINUITY.Distributed_Semantic_Fragmentation_Detected THEN
    L_Semantic_Valid := FALSE;
    L_Error_Code := 31006;
    L_Error_Text := 'Distributed semantic fragmentation detected';
END_IF;

// Intent continuity validation.
IF L_Semantic_Valid
AND NOT GVL_SEMANTIC_CONTINUITY.Declared_System_Intent_Valid THEN
    L_Semantic_Valid := FALSE;
    L_Error_Code := 31010;
    L_Error_Text := 'Declared system intent invalid';
END_IF;

IF L_Semantic_Valid
AND NOT GVL_SEMANTIC_CONTINUITY.Runtime_Goal_Alignment_Valid THEN
    L_Semantic_Valid := FALSE;
    L_Error_Code := 31011;
    L_Error_Text := 'Runtime goal alignment invalid';
END_IF;

IF L_Semantic_Valid
AND NOT GVL_SEMANTIC_CONTINUITY.Optimization_Boundary_Valid THEN
    L_Semantic_Valid := FALSE;
    L_Error_Code := 31012;
    L_Error_Text := 'Optimization boundary invalid';
END_IF;

IF L_Semantic_Valid
AND NOT GVL_SEMANTIC_CONTINUITY.Autonomous_Adjustment_Valid THEN
    L_Semantic_Valid := FALSE;
    L_Error_Code := 31013;
    L_Error_Text := 'Autonomous adjustment invalid';
END_IF;

IF L_Semantic_Valid THEN
    GVL_SEMANTIC_CONTINUITY.Semantic_Continuity_Valid := TRUE;
    GVL_SEMANTIC_CONTINUITY.Semantic_Continuity_Granted := TRUE;
    GVL_SEMANTIC_CONTINUITY.Semantic_Continuity_Quarantine_Active := FALSE;

    GVL_SEMANTIC_CONTINUITY.Operator_Intent_Coherent := TRUE;
    GVL_SEMANTIC_CONTINUITY.Policy_Intent_Coherent := TRUE;
    GVL_SEMANTIC_CONTINUITY.Adaptive_Behavior_Coherent := TRUE;
    GVL_SEMANTIC_CONTINUITY.Recovery_Intent_Coherent := TRUE;
    GVL_SEMANTIC_CONTINUITY.Distributed_Semantic_Coherent := TRUE;

    GVL_SEMANTIC_CONTINUITY.Semantic_Continuity_Epoch :=
        GVL_RUNTIME_RESOURCE_AUTHORITY.Runtime_Resource_Authority_Epoch;

    GVL_SEMANTIC_CONTINUITY.Semantic_Continuity_Epoch_Coherent := TRUE;

    GVL_SEMANTIC_CONTINUITY.Semantic_Last_Update_MS := L_Now_MS;
    GVL_SEMANTIC_CONTINUITY.Semantic_Lease_Expired := FALSE;

    GVL_SEMANTIC_CONTINUITY.Semantic_Last_Error_Code := 0;
    GVL_SEMANTIC_CONTINUITY.Semantic_Last_Error_Text := '';
ELSE
    GVL_SEMANTIC_CONTINUITY.Semantic_Continuity_Valid := FALSE;
    GVL_SEMANTIC_CONTINUITY.Semantic_Continuity_Granted := FALSE;
    GVL_SEMANTIC_CONTINUITY.Semantic_Continuity_Quarantine_Active := TRUE;

    GVL_SEMANTIC_CONTINUITY.Semantic_Lease_Expired := TRUE;

    GVL_SEMANTIC_CONTINUITY.Semantic_Last_Error_Code :=
        L_Error_Code;

    GVL_SEMANTIC_CONTINUITY.Semantic_Last_Error_Text :=
        L_Error_Text;

    GVL_SEMANTIC_CONTINUITY.Semantic_Invalidation_Count :=
        GVL_SEMANTIC_CONTINUITY.Semantic_Invalidation_Count + 1;
END_IF;
          
END_PROGRAM

PROGRAM PRG_System_Diagnostics_Ext
  VAR
    L_Error_Heating : BOOL;
    L_Error_Safety : BOOL;
    L_Error_IO : BOOL;
    L_Delta_Time : REAL;
    L_Now : UDINT;
    L_Last : UDINT;
    L_Cycle_MS : UDINT;
    L_Prev_Overrun : BOOL;
    L_Prev_Critical : BOOL;
    fbLog : FB_LogEvent;
  END_VAR

            L_Now := GVL_TIME_SERVICE.G_Now_MS;
L_Last := GVL_DIAGNOSTICS_EXT.G_Last_Update_Time;

// ===============================
// CYCLE INTERVAL MEASUREMENT
// ===============================
IF L_Last = 0 THEN
    L_Cycle_MS := GVL_DIAGNOSTICS_EXT.G_Cycle_Expected_MS;
ELSE
    IF L_Now >= L_Last THEN
        L_Cycle_MS := L_Now - L_Last;
    ELSE
        L_Cycle_MS := (4294967295 - L_Last) + L_Now + 1;
    END_IF;
END_IF;

GVL_DIAGNOSTICS_EXT.G_Last_Update_Time := L_Now;
GVL_DIAGNOSTICS_EXT.G_Cycle_Last_MS := L_Cycle_MS;

// min/max
IF (GVL_DIAGNOSTICS_EXT.G_Cycle_Min_MS = 0) OR (L_Cycle_MS < GVL_DIAGNOSTICS_EXT.G_Cycle_Min_MS) THEN
    GVL_DIAGNOSTICS_EXT.G_Cycle_Min_MS := L_Cycle_MS;
END_IF;

IF L_Cycle_MS > GVL_DIAGNOSTICS_EXT.G_Cycle_Max_MS THEN
    GVL_DIAGNOSTICS_EXT.G_Cycle_Max_MS := L_Cycle_MS;
END_IF;

// average (incremental)
GVL_DIAGNOSTICS_EXT.G_Cycle_Sample_Count := GVL_DIAGNOSTICS_EXT.G_Cycle_Sample_Count + 1;
GVL_DIAGNOSTICS_EXT.G_Cycle_Avg_MS :=
    GVL_DIAGNOSTICS_EXT.G_Cycle_Avg_MS +
    (UDINT_TO_REAL(L_Cycle_MS) - GVL_DIAGNOSTICS_EXT.G_Cycle_Avg_MS) /
    UDINT_TO_REAL(GVL_DIAGNOSTICS_EXT.G_Cycle_Sample_Count);

// ===============================
// OVERRUN / CRITICAL DETECTION
// ===============================
GVL_DIAGNOSTICS_EXT.G_Cycle_Overrun_Active := (L_Cycle_MS > GVL_DIAGNOSTICS_EXT.G_Cycle_Warning_MS);
GVL_DIAGNOSTICS_EXT.G_Cycle_Critical_Active := (L_Cycle_MS > GVL_DIAGNOSTICS_EXT.G_Cycle_Critical_MS);

IF GVL_DIAGNOSTICS_EXT.G_Cycle_Overrun_Active THEN
    GVL_DIAGNOSTICS_EXT.G_Cycle_Overrun_Count := GVL_DIAGNOSTICS_EXT.G_Cycle_Overrun_Count + 1;
    GVL_DIAGNOSTICS_EXT.G_Cycle_Last_Overrun_MS := L_Cycle_MS;
    GVL_DIAGNOSTICS_EXT.G_Cycle_Last_Overrun_Time_MS := L_Now;
END_IF;

IF GVL_DIAGNOSTICS_EXT.G_Cycle_Critical_Active THEN
    GVL_DIAGNOSTICS_EXT.G_Cycle_Critical_Count := GVL_DIAGNOSTICS_EXT.G_Cycle_Critical_Count + 1;
END_IF;

// edge logging
IF GVL_DIAGNOSTICS_EXT.G_Cycle_Overrun_Active AND NOT L_Prev_Overrun THEN
    fbLog(
        VI_Event_Type := 2001,
        VI_Timestamp := L_Now,
        VI_Param1 := L_Cycle_MS,
        VI_Param2 := GVL_DIAGNOSTICS_EXT.G_Cycle_Overrun_Count
    );
END_IF;

IF GVL_DIAGNOSTICS_EXT.G_Cycle_Critical_Active AND NOT L_Prev_Critical THEN
    fbLog(
        VI_Event_Type := 2002,
        VI_Timestamp := L_Now,
        VI_Param1 := L_Cycle_MS,
        VI_Param2 := GVL_DIAGNOSTICS_EXT.G_Cycle_Critical_Count
    );
END_IF;

L_Prev_Overrun := GVL_DIAGNOSTICS_EXT.G_Cycle_Overrun_Active;
L_Prev_Critical := GVL_DIAGNOSTICS_EXT.G_Cycle_Critical_Active;

// ===============================
// EXISTING HEALTH LOGIC
// ===============================
IF L_Last = 0 THEN
    L_Delta_Time := 0.1;
ELSE
    L_Delta_Time := UDINT_TO_REAL(L_Cycle_MS) / 1000.0;
END_IF;

L_Error_Heating := GVL_STATE.G_Heating_Subsystem_Degraded;

// Extended diagnostics must use authoritative safety truth and latches,
// not stale projected GVL_STATE.G_Safety_*_Alarm compatibility fields.
L_Error_Safety :=
    GVL_HEALTH_BRIDGE.G_Gas_Detected OR
    GVL_HEALTH_BRIDGE.G_CO_Alarm_Level OR
    GVL_HEALTH_BRIDGE.G_Leak_Detected OR
    GVL_HEALTH_BRIDGE.G_Smoke_Detected OR
    GVL_STATE.G_Safety_Gas_Latched OR
    GVL_STATE.G_Safety_Leak_Latched OR
    GVL_STATE.G_Safety_Smoke_Latched;

L_Error_IO := GVL_STATE.G_Heating_IO_Fault;

IF L_Error_Heating THEN
    GVL_DIAGNOSTICS_EXT.G_Error_Count_Heating := GVL_DIAGNOSTICS_EXT.G_Error_Count_Heating + 1;
    GVL_DIAGNOSTICS_EXT.G_Last_Error_Time_Heating := L_Now;
    GVL_DIAGNOSTICS_EXT.G_Health_Heating := GVL_DIAGNOSTICS_EXT.G_Health_Heating - (0.5 * L_Delta_Time);
ELSE
    GVL_DIAGNOSTICS_EXT.G_Health_Heating := GVL_DIAGNOSTICS_EXT.G_Health_Heating + (0.1 * L_Delta_Time);
END_IF;

IF L_Error_Safety THEN
    GVL_DIAGNOSTICS_EXT.G_Error_Count_Safety := GVL_DIAGNOSTICS_EXT.G_Error_Count_Safety + 1;
    GVL_DIAGNOSTICS_EXT.G_Last_Error_Time_Safety := L_Now;
    GVL_DIAGNOSTICS_EXT.G_Health_Safety := GVL_DIAGNOSTICS_EXT.G_Health_Safety - (1.0 * L_Delta_Time);
ELSE
    GVL_DIAGNOSTICS_EXT.G_Health_Safety := GVL_DIAGNOSTICS_EXT.G_Health_Safety + (0.2 * L_Delta_Time);
END_IF;

IF L_Error_IO THEN
    GVL_DIAGNOSTICS_EXT.G_Error_Count_IO := GVL_DIAGNOSTICS_EXT.G_Error_Count_IO + 1;
    GVL_DIAGNOSTICS_EXT.G_Last_Error_Time_IO := L_Now;
    GVL_DIAGNOSTICS_EXT.G_Health_IO := GVL_DIAGNOSTICS_EXT.G_Health_IO - (0.5 * L_Delta_Time);
ELSE
    GVL_DIAGNOSTICS_EXT.G_Health_IO := GVL_DIAGNOSTICS_EXT.G_Health_IO + (0.1 * L_Delta_Time);
END_IF;

// clamp
IF GVL_DIAGNOSTICS_EXT.G_Health_Heating < 0.0 THEN GVL_DIAGNOSTICS_EXT.G_Health_Heating := 0.0; END_IF;
IF GVL_DIAGNOSTICS_EXT.G_Health_Heating > 1.0 THEN GVL_DIAGNOSTICS_EXT.G_Health_Heating := 1.0; END_IF;

IF GVL_DIAGNOSTICS_EXT.G_Health_Safety < 0.0 THEN GVL_DIAGNOSTICS_EXT.G_Health_Safety := 0.0; END_IF;
IF GVL_DIAGNOSTICS_EXT.G_Health_Safety > 1.0 THEN GVL_DIAGNOSTICS_EXT.G_Health_Safety := 1.0; END_IF;

IF GVL_DIAGNOSTICS_EXT.G_Health_IO < 0.0 THEN GVL_DIAGNOSTICS_EXT.G_Health_IO := 0.0; END_IF;
IF GVL_DIAGNOSTICS_EXT.G_Health_IO > 1.0 THEN GVL_DIAGNOSTICS_EXT.G_Health_IO := 1.0; END_IF;
          
END_PROGRAM

PROGRAM PRG_HA_Session_Replication

            // ======================================================
// HA SESSION REPLICATION
// ======================================================
// Dedicated HA/session replication boundary.
//
// Purpose:
// replicate canonical peer-session state through isolated
// HA replication surface.
//
// Current implementation:
// bounded loopback foundation.
//
// Future implementations may replace this with:
// - SysCom HA channel
// - shared-memory replication
// - dedicated Ethernet HA link
// - deterministic fieldbus synchronization
//
// without changing distributed governors.
// ======================================================

IF NOT GVL_HA_SESSION_REPLICATION.HA_Replication_Enabled THEN
    GVL_HA_SESSION_REPLICATION.HA_Channel_Healthy := FALSE;
    RETURN;
END_IF;

// ------------------------------------------------------
// Canonical session export replication.
// ------------------------------------------------------

GVL_HA_SESSION_REPLICATION.HA_Remote_Session_Valid :=
    GVL_PEER_SESSION.Remote_Session_Valid;

GVL_HA_SESSION_REPLICATION.HA_Remote_Last_Refresh_MS :=
    GVL_PEER_SESSION.Remote_Last_Refresh_MS;

GVL_HA_SESSION_REPLICATION.HA_Remote_Runtime_Epoch :=
    GVL_PEER_SESSION.Remote_Runtime_Epoch;

GVL_HA_SESSION_REPLICATION.HA_Remote_Snapshot_Epoch :=
    GVL_PEER_SESSION.Remote_Snapshot_Epoch;

GVL_HA_SESSION_REPLICATION.HA_Remote_Boot_Generation :=
    GVL_PEER_SESSION.Remote_Boot_Generation;

GVL_HA_SESSION_REPLICATION.HA_Remote_Fencing_Token :=
    GVL_PEER_SESSION.Remote_Fencing_Token;

GVL_HA_SESSION_REPLICATION.HA_Remote_Publication_Allowed :=
    GVL_PEER_SESSION.Remote_Publication_Allowed;

GVL_HA_SESSION_REPLICATION.HA_Remote_Runtime_Healthy :=
    GVL_PEER_SESSION.Remote_Runtime_Healthy;

GVL_HA_SESSION_REPLICATION.HA_Last_TX_MS :=
    GVL_STATUS.G_System_Time_MS;

GVL_HA_SESSION_REPLICATION.HA_Last_RX_MS :=
    GVL_STATUS.G_System_Time_MS;

GVL_HA_SESSION_REPLICATION.HA_Channel_Healthy := TRUE;

// >>> BULK_SYNC_ANCHOR: PRG_HA_Session_Replication <<<
          
END_PROGRAM

PROGRAM PRG_Modbus_RTU_SysCom_Backend
  VAR
    FB_Backend : FB_Modbus_RTU_SysCom_Backend;
  END_VAR

            FB_Backend(
    VI_Enable := GVL_CONFIG.G_OpenTherm_Enabled,
    VI_System_Time_MS := GVL_STATUS.G_System_Time_MS
);
          
END_PROGRAM

PROGRAM PRG_Mode_Manager
  VAR
    fbMode : FB_Mode_Manager;
    L_Last_Mode : E_Behavior_Mode := BEHAVIOR_HOME;
  END_VAR

            fbMode(
    VI_Is_Night := GVL_STATUS.G_Is_Night,
    VI_Away_Request := GVL_MODE.G_Away_Request OR GVL_PRESENCE.G_Auto_Away_Request,
    VI_Maintenance_Request := GVL_MODE.G_Maintenance_Request,
    VI_System_Time_MS := GVL_STATUS.G_System_Time_MS
);

GVL_MODE.G_Current_Behavior_Mode := fbMode.VO_Mode;
GVL_MODE.G_Mode_Code := fbMode.VO_Mode_Code;

IF L_Last_Mode <> fbMode.VO_Mode THEN
    GVL_MODE.G_Mode_Last_Change_TS := GVL_STATUS.G_System_Time_MS;
    L_Last_Mode := fbMode.VO_Mode;
END_IF;
          
END_PROGRAM

PROGRAM PRG_System_Coordinator
  VAR
    fbCoord : FB_System_Coordinator;
  END_VAR

            fbCoord(
    VI_Fire_Latched := GVL_STATE.G_Safety_Smoke_Latched,
    VI_Gas_Latched := GVL_STATE.G_Safety_Gas_Latched,
    VI_Leak_Latched := GVL_STATE.G_Safety_Leak_Latched,
    VI_IO_Degraded := NOT GVL_STATUS.G_IO_Modules_Online[1],
    VI_Ownership_Violation := FALSE,
    VI_Behavior_Mode := GVL_MODE.G_Current_Behavior_Mode
);

GVL_SYSTEM_COORDINATION.G_Block_Heating := fbCoord.VO_Block_Heating OR GVL_HEATING_POLICY.G_Policy_Block_Heating_Request;
GVL_SYSTEM_COORDINATION.G_Block_Ventilation := fbCoord.VO_Block_Ventilation;
GVL_SYSTEM_COORDINATION.G_Block_Lighting_Override := fbCoord.VO_Block_Lighting;
GVL_SYSTEM_COORDINATION.G_Block_Sockets_Override := fbCoord.VO_Block_Sockets;

GVL_SYSTEM_COORDINATION.G_System_Degraded := fbCoord.VO_System_Degraded;
GVL_SYSTEM_COORDINATION.G_Coordination_Code := fbCoord.VO_Code;
          
END_PROGRAM

PROGRAM PRG_Time_Monotonic_Governor
  VAR
    L_Now_MS : UDINT;
    L_Delta_MS : UDINT;
    L_Time_Valid : BOOL := TRUE;
    L_Error_Code : UDINT := 0;
    L_Error_Text : STRING(160) := '';
  END_VAR

            L_Now_MS := GVL_STATUS.G_System_Time_MS;
L_Time_Valid := TRUE;
L_Error_Code := 0;
L_Error_Text := '';

// ======================================================
// MONOTONIC TIME GOVERNOR
// ======================================================
// Creates monotonic time authority semantics.
// Prevents rollback/reboot resurrection.
// ======================================================

// First initialization.
IF NOT GVL_TIME_MONOTONIC.Monotonic_Time_Initialized THEN
    GVL_TIME_MONOTONIC.Monotonic_Time_Initialized := TRUE;
    GVL_TIME_MONOTONIC.Boot_Generation_ID := GVL_TIME_MONOTONIC.Boot_Generation_ID + 1;
    GVL_TIME_MONOTONIC.Startup_Quarantine_Active := TRUE;
    GVL_TIME_MONOTONIC.Startup_Quarantine_Start_MS := L_Now_MS;
    GVL_TIME_MONOTONIC.Last_Monotonic_Time_MS := L_Now_MS;
END_IF;

GVL_TIME_MONOTONIC.Time_Rollback_Detected := FALSE;
GVL_TIME_MONOTONIC.Time_Overflow_Detected := FALSE;
GVL_TIME_MONOTONIC.Retained_Time_Invalid := FALSE;
GVL_TIME_MONOTONIC.Startup_Quarantine_Release_Allowed := FALSE;

// Rollback detection.
IF L_Now_MS < GVL_TIME_MONOTONIC.Last_Monotonic_Time_MS THEN
    L_Time_Valid := FALSE;
    L_Error_Code := 8000;
    L_Error_Text := 'Monotonic rollback detected';

    GVL_TIME_MONOTONIC.Time_Rollback_Detected := TRUE;
    GVL_TIME_MONOTONIC.Retained_Time_Invalid := TRUE;
END_IF;

// Overflow / invalid delta detection.
L_Delta_MS := L_Now_MS - GVL_TIME_MONOTONIC.Last_Monotonic_Time_MS;

IF L_Time_Valid AND (L_Delta_MS > 60000) THEN
    L_Time_Valid := FALSE;
    L_Error_Code := 8001;
    L_Error_Text := 'Monotonic delta overflow';

    GVL_TIME_MONOTONIC.Time_Overflow_Detected := TRUE;
END_IF;

// Startup quarantine governance.
IF GVL_TIME_MONOTONIC.Startup_Quarantine_Active THEN
    IF (L_Now_MS - GVL_TIME_MONOTONIC.Startup_Quarantine_Start_MS) >= GVL_TIME_MONOTONIC.Startup_Quarantine_Timeout_MS THEN
        GVL_TIME_MONOTONIC.Startup_Quarantine_Active := FALSE;
        GVL_TIME_MONOTONIC.Startup_Quarantine_Release_Allowed := TRUE;
    ELSE
        L_Time_Valid := FALSE;

        IF L_Error_Code = 0 THEN
            L_Error_Code := 8002;
            L_Error_Text := 'Startup quarantine active';
        END_IF;
    END_IF;
END_IF;

// Publish monotonic authority state.
IF L_Time_Valid THEN
    GVL_TIME_MONOTONIC.Monotonic_Epoch := GVL_TIME_MONOTONIC.Monotonic_Epoch + 1;
    GVL_TIME_MONOTONIC.Monotonic_Time_Valid := TRUE;
    GVL_TIME_MONOTONIC.Last_Validated_Time_MS := L_Now_MS;
    GVL_TIME_MONOTONIC.Last_Monotonic_Time_MS := L_Now_MS;

    GVL_TIME_MONOTONIC.Monotonic_Last_Error_Code := 0;
    GVL_TIME_MONOTONIC.Monotonic_Last_Error_Text := '';
ELSE
    GVL_TIME_MONOTONIC.Monotonic_Time_Valid := FALSE;
    GVL_TIME_MONOTONIC.Monotonic_Last_Error_Code := L_Error_Code;
    GVL_TIME_MONOTONIC.Monotonic_Last_Error_Text := L_Error_Text;

    GVL_TIME_MONOTONIC.Monotonic_Invalidation_Count := GVL_TIME_MONOTONIC.Monotonic_Invalidation_Count + 1;
END_IF;
          
END_PROGRAM

PROGRAM PRG_Semantic_Drift_Observability_Governor

            // PASSIVE OBSERVABILITY ONLY

GVL_SEMANTIC_DRIFT_OBSERVABILITY_FABRIC.Semantic_Continuity_Observed :=
    GVL_PASSIVE_RUNTIME_VERIFICATION_FABRIC.Runtime_Verification_Consistency_Valid;

GVL_SEMANTIC_DRIFT_OBSERVABILITY_FABRIC.Semantic_Projection_Consistency_Observed := TRUE;
GVL_SEMANTIC_DRIFT_OBSERVABILITY_FABRIC.Distributed_Semantic_Alignment_Observed := TRUE;
          
END_PROGRAM

PROGRAM PRG_Ventilation
  VAR
    fbVentilationManager : FB_Ventilation_System_Manager;
    fbVentProjection : FB_Vent_Output_Projection;
    L_i : INT;
    L_Supply_Fans_Byte : ARRAY[1..GVL_CONSTANTS.C_MAX_SUPPLY_FANS] OF BYTE;
    L_Exhaust_Fans_Byte : ARRAY[1..GVL_CONSTANTS.C_MAX_EXHAUST_FANS] OF BYTE;
    L_Wet_Zone_Active : ARRAY[1..GVL_CONSTANTS.C_MAX_WET_ZONES] OF BOOL;
    L_Vent_PV3_Boost_Req : BOOL;
    L_Supply_100_Req : BOOL;
    L_Exhaust_100_Req : BOOL;
    L_Supply_80_Req : BOOL;
    L_Vent_Stop_Req : BOOL;
    L_Distributed_Execute_Allowed : BOOL;
    L_Distributed_Projection_Allowed : BOOL;
    L_Fire_Smoke_Override : BOOL;
  END_VAR

            // Distributed runtime governance.
// FIRE smoke extraction semantics remain authoritative.
L_Distributed_Execute_Allowed :=
    GVL_Distributed_Execution_Gates.G_Can_Execute;

L_Distributed_Projection_Allowed :=
    GVL_Distributed_Execution_Gates.G_Can_Own_Projection;

L_Fire_Smoke_Override :=
    GVL_COMMAND_SHADOW.G_Vent_Smoke_Exhaust;

// Wet-zone adapter
FOR L_i := 1 TO GVL_CONSTANTS.C_MAX_WET_ZONES DO
    L_Wet_Zone_Active[L_i] := FALSE;
END_FOR;

IF GVL_STATUS.G_Wet_Zone_Light_Active THEN
    L_Wet_Zone_Active[1] := TRUE;
END_IF;

// === Ventilation Inputs (from arbitration only) ===
L_Vent_PV3_Boost_Req := GVL_COMMAND_SHADOW.G_Vent_PV3_Boost;
L_Supply_100_Req := GVL_COMMAND_SHADOW.G_Supply_100_Req;
L_Exhaust_100_Req := GVL_COMMAND_SHADOW.G_Exhaust_100_Req;
L_Supply_80_Req := GVL_COMMAND_SHADOW.G_Supply_80_Req;
L_Vent_Stop_Req := GVL_COMMAND_SHADOW.G_Vent_Stop;

IF L_Distributed_Execute_Allowed THEN

    // Ventilation control (execution core)
    fbVentilationManager(
        VI_System_Time_MS := GVL_STATUS.G_System_Time_MS,
        VI_IsActivePLC := GVL_STATUS.G_Is_Active_PLC,
        VI_Outdoor_Temp := GVL_STATE.G_Outdoor_Temp,
        VI_Supply_Temps := GVL_STATE.G_Supply_Temps,
        VI_Room_Temps := GVL_STATE.G_Room_Temps,
        VI_Room_Humidities := GVL_STATE.G_Room_Hum,
        VI_Room_CO2 := GVL_STATE.G_Room_CO2,
        VI_Current_Scenario := GVL_STATUS.G_Current_Scenario,
        VI_System_Mode := GVL_STATE.G_System_Mode,
        VI_Config := GVL_CONFIG.G_HMI_Vent_Global_Config,
        VI_Fire_Alarm := GVL_STATE.G_Safety_Smoke_Latched,
        VI_Gas_Alarm := GVL_STATE.G_Safety_Gas_Latched,
        VI_PV3_Boost_Req := L_Vent_PV3_Boost_Req,
        VI_Supply_100_Req := L_Supply_100_Req,
        VI_Exhaust_100_Req := L_Exhaust_100_Req,
        VI_Supply_80_Req := L_Supply_80_Req,
        VI_Vent_Stop := L_Vent_Stop_Req,
        VI_IO_Modules_Online := GVL_STATUS.G_IO_Modules_Online,
        VI_Wet_Zone_Active := L_Wet_Zone_Active,
        VI_Rule_Actions := GVL_STATE.G_Rule_Actions,
        VO_Supply_Fans => L_Supply_Fans_Byte,
        VO_Exhaust_Fans => L_Exhaust_Fans_Byte,
        VO_Heater_Power => GVL_STATE.G_Vent_Heater_Power,
        VO_Status_Msg => GVL_STATUS.G_Vent_Status_Msg,
        VO_Ventilation_IO_Fault => GVL_STATE.G_Ventilation_IO_Fault,
        VO_Ventilation_Subsystem_Degraded => GVL_STATE.G_Ventilation_Subsystem_Degraded
    );

END_IF;

// ==============================
// SMOKE EXHAUST OVERRIDE
// ==============================
// FIRE smoke extraction must remain authoritative
// even during distributed degradation.
IF L_Fire_Smoke_Override THEN

    FOR L_i := 1 TO GVL_CONSTANTS.C_MAX_EXHAUST_FANS DO
        L_Exhaust_Fans_Byte[L_i] := 100;
    END_FOR;

    FOR L_i := 1 TO GVL_CONSTANTS.C_MAX_SUPPLY_FANS DO
        L_Supply_Fans_Byte[L_i] := 0;
    END_FOR;

END_IF;

// Distributed projection restriction.
IF NOT L_Distributed_Projection_Allowed
   AND NOT L_Fire_Smoke_Override THEN

    FOR L_i := 1 TO GVL_CONSTANTS.C_MAX_EXHAUST_FANS DO
        L_Exhaust_Fans_Byte[L_i] := 0;
    END_FOR;

    FOR L_i := 1 TO GVL_CONSTANTS.C_MAX_SUPPLY_FANS DO
        L_Supply_Fans_Byte[L_i] := 0;
    END_FOR;

END_IF;

// === OUTPUT PROJECTION ===
fbVentProjection(
    VI_Supply_Fans := L_Supply_Fans_Byte,
    VI_Exhaust_Fans := L_Exhaust_Fans_Byte
);

// >>> BULK_SYNC_ANCHOR: PRG_Ventilation <<<
          
END_PROGRAM

PROGRAM PRG_Recovery_Domain

            // SEMANTIC DOMAIN WRAPPER
// PRESERVES ORIGINAL EXECUTION ORDER

PRG_Recovery_Cleanup_Governor();
PRG_Deterministic_Recovery_Path_Governor();
PRG_Recovery_Ordering_Integrity_Governor();
PRG_Recovery_Reactivation_Control_Governor();
PRG_Authority_Resurrection_Boundary_Governor();

PRG_Energy_Resurrection_Boundary_Governor();
PRG_Physical_Deadlock_Resolution_Governor();
          
END_PROGRAM

PROGRAM PRG_Operational_Intelligence_Governor

            // PASSIVE OPERATIONAL INTELLIGENCE
// NO EXECUTION MUTATION
// NO AUTHORITY MUTATION

GVL_OPERATIONAL_INTELLIGENCE_FABRIC.Operational_Reasoning_Consistency_Valid :=
    GVL_RUNTIME_TRANSITION_SYSTEM.Runtime_Transition_Legal;

GVL_OPERATIONAL_INTELLIGENCE_FABRIC.Runtime_Causal_Projection_Valid :=
    GVL_TEMPORAL_CAUSALITY_CLOSURE_FABRIC.Temporal_Causality_Coherent;

GVL_OPERATIONAL_INTELLIGENCE_FABRIC.Distributed_Operational_Context_Valid :=
    GVL_DISTRIBUTED_SAFETY_REALITY_CONSENSUS_FABRIC.Distributed_Safety_Consensus_Valid;

IF GVL_RUNTIME_TRANSITION_SYSTEM.Illegal_Runtime_Transition_Observed THEN
    GVL_OPERATIONAL_INTELLIGENCE_FABRIC.Active_Degradation_Cause_Available := TRUE;
END_IF;

IF GVL_RUNTIME_TRANSITION_SYSTEM.Recovery_Without_Lineage_Observed THEN
    GVL_OPERATIONAL_INTELLIGENCE_FABRIC.Recovery_Blocker_Observed := TRUE;
END_IF;
          
END_PROGRAM

PROGRAM PRG_Physical_Transaction_Governor
  VAR
    L_Now_MS : UDINT;
    L_Transaction_Valid : BOOL := TRUE;
    L_Error_Code : UDINT := 0;
    L_Error_Text : STRING(160) := '';
  END_VAR

            L_Now_MS := GVL_STATUS.G_System_Time_MS;
L_Transaction_Valid := TRUE;
L_Error_Code := 0;
L_Error_Text := '';

// Fail-safe defaults.
GVL_PHYSICAL_TRANSACTION.Physical_Transaction_Valid := FALSE;
GVL_PHYSICAL_TRANSACTION.Physical_Transaction_Granted := FALSE;
GVL_PHYSICAL_TRANSACTION.Physical_Transaction_Quarantine_Active := TRUE;

GVL_PHYSICAL_TRANSACTION.All_Actuators_Converged := FALSE;
GVL_PHYSICAL_TRANSACTION.Cross_Actuator_Epoch_Coherent := FALSE;
GVL_PHYSICAL_TRANSACTION.Distributed_Actuation_Coherent := FALSE;
GVL_PHYSICAL_TRANSACTION.Stable_Plant_State_Confirmed := FALSE;

// Bind transaction epochs.
GVL_PHYSICAL_TRANSACTION.Physical_Transaction_Command_Epoch :=
    GVL_ACTUATION_AUTHORITY.Actuation_Command_Epoch;

GVL_PHYSICAL_TRANSACTION.Physical_Transaction_ACK_Epoch :=
    GVL_ACTUATION_AUTHORITY.Field_ACK_Epoch;

IF GVL_PHYSICAL_TRANSACTION.Physical_Transaction_Command_Epoch <>
   GVL_PHYSICAL_TRANSACTION.Physical_Transaction_ACK_Epoch THEN

    GVL_PHYSICAL_TRANSACTION.Cross_Actuator_Convergence_Skew := TRUE;

    L_Transaction_Valid := FALSE;
    L_Error_Code := 27000;
    L_Error_Text := 'Physical transaction epoch skew detected';
END_IF;

// Ordering race detection.
IF L_Transaction_Valid
AND GVL_PHYSICAL_TRANSACTION.Pump_Valve_Ordering_Race_Detected THEN
    L_Transaction_Valid := FALSE;
    L_Error_Code := 27001;
    L_Error_Text := 'Pump/valve ordering race detected';
END_IF;

// Brownout / rollback protection.
IF L_Transaction_Valid
AND GVL_PHYSICAL_TRANSACTION.Distributed_Actuator_Rollback_Detected THEN
    L_Transaction_Valid := FALSE;
    L_Error_Code := 27002;
    L_Error_Text := 'Distributed actuator rollback detected';
END_IF;

IF L_Transaction_Valid
AND GVL_PHYSICAL_TRANSACTION.Brownout_Partial_Switching_Detected THEN
    L_Transaction_Valid := FALSE;
    L_Error_Code := 27003;
    L_Error_Text := 'Brownout partial switching detected';
END_IF;

IF L_Transaction_Valid
AND GVL_PHYSICAL_TRANSACTION.Transaction_Timeout_Detected THEN
    L_Transaction_Valid := FALSE;
    L_Error_Code := 27004;
    L_Error_Text := 'Physical transaction timeout detected';
END_IF;

IF L_Transaction_Valid
AND GVL_PHYSICAL_TRANSACTION.Partial_Plant_Transition_Detected THEN
    L_Transaction_Valid := FALSE;
    L_Error_Code := 27005;
    L_Error_Text := 'Partial plant transition detected';
END_IF;

// All actuator transitions required.
IF L_Transaction_Valid
AND NOT GVL_PHYSICAL_TRANSACTION.Valve_Transition_Confirmed THEN
    L_Transaction_Valid := FALSE;
    L_Error_Code := 27010;
    L_Error_Text := 'Valve transition confirmation missing';
END_IF;

IF L_Transaction_Valid
AND NOT GVL_PHYSICAL_TRANSACTION.Pump_Transition_Confirmed THEN
    L_Transaction_Valid := FALSE;
    L_Error_Code := 27011;
    L_Error_Text := 'Pump transition confirmation missing';
END_IF;

IF L_Transaction_Valid
AND NOT GVL_PHYSICAL_TRANSACTION.Damper_Transition_Confirmed THEN
    L_Transaction_Valid := FALSE;
    L_Error_Code := 27012;
    L_Error_Text := 'Damper transition confirmation missing';
END_IF;

IF L_Transaction_Valid
AND NOT GVL_PHYSICAL_TRANSACTION.Relay_Bank_Transition_Confirmed THEN
    L_Transaction_Valid := FALSE;
    L_Error_Code := 27013;
    L_Error_Text := 'Relay bank transition confirmation missing';
END_IF;

// Stable plant convergence required.
IF L_Transaction_Valid
AND NOT GVL_PHYSICAL_TRANSACTION.Flow_Stabilization_Confirmed THEN
    L_Transaction_Valid := FALSE;
    L_Error_Code := 27020;
    L_Error_Text := 'Flow stabilization missing';
END_IF;

IF L_Transaction_Valid
AND NOT GVL_PHYSICAL_TRANSACTION.Pressure_Stabilization_Confirmed THEN
    L_Transaction_Valid := FALSE;
    L_Error_Code := 27021;
    L_Error_Text := 'Pressure stabilization missing';
END_IF;

IF L_Transaction_Valid
AND NOT GVL_PHYSICAL_TRANSACTION.Thermal_Response_Confirmed THEN
    L_Transaction_Valid := FALSE;
    L_Error_Code := 27022;
    L_Error_Text := 'Thermal response confirmation missing';
END_IF;

IF L_Transaction_Valid
AND NOT GVL_PHYSICAL_TRANSACTION.Electrical_Load_Stabilized THEN
    L_Transaction_Valid := FALSE;
    L_Error_Code := 27023;
    L_Error_Text := 'Electrical load stabilization missing';
END_IF;

IF L_Transaction_Valid THEN
    GVL_PHYSICAL_TRANSACTION.Physical_Transaction_Valid := TRUE;
    GVL_PHYSICAL_TRANSACTION.Physical_Transaction_Granted := TRUE;
    GVL_PHYSICAL_TRANSACTION.Physical_Transaction_Quarantine_Active := FALSE;

    GVL_PHYSICAL_TRANSACTION.All_Actuators_Converged := TRUE;
    GVL_PHYSICAL_TRANSACTION.Cross_Actuator_Epoch_Coherent := TRUE;
    GVL_PHYSICAL_TRANSACTION.Distributed_Actuation_Coherent := TRUE;
    GVL_PHYSICAL_TRANSACTION.Stable_Plant_State_Confirmed := TRUE;

    GVL_PHYSICAL_TRANSACTION.Physical_Transaction_Epoch :=
        GVL_PHYSICAL_TRANSACTION.Physical_Transaction_Command_Epoch;

    GVL_PHYSICAL_TRANSACTION.Physical_Transaction_Last_Update_MS :=
        L_Now_MS;

    GVL_PHYSICAL_TRANSACTION.Physical_Transaction_Lease_Expired := FALSE;

    GVL_PHYSICAL_TRANSACTION.Physical_Transaction_Last_Error_Code := 0;
    GVL_PHYSICAL_TRANSACTION.Physical_Transaction_Last_Error_Text := '';
ELSE
    GVL_PHYSICAL_TRANSACTION.Physical_Transaction_Valid := FALSE;
    GVL_PHYSICAL_TRANSACTION.Physical_Transaction_Granted := FALSE;
    GVL_PHYSICAL_TRANSACTION.Physical_Transaction_Quarantine_Active := TRUE;

    GVL_PHYSICAL_TRANSACTION.Physical_Transaction_Lease_Expired := TRUE;

    GVL_PHYSICAL_TRANSACTION.Physical_Transaction_Last_Error_Code :=
        L_Error_Code;

    GVL_PHYSICAL_TRANSACTION.Physical_Transaction_Last_Error_Text :=
        L_Error_Text;

    GVL_PHYSICAL_TRANSACTION.Physical_Transaction_Invalidation_Count :=
        GVL_PHYSICAL_TRANSACTION.Physical_Transaction_Invalidation_Count + 1;
END_IF;
          
END_PROGRAM

PROGRAM PRG_Distributed_Commit_Governor
  VAR
    L_Now_MS : UDINT;
    L_Delta_MS : UDINT;
    L_Commit_Valid : BOOL := TRUE;
    L_Error_Code : UDINT := 0;
    L_Error_Text : STRING(160) := '';
    L_Peer_Session_Active : BOOL := FALSE;
    L_Publication_Authority_Allowed : BOOL;
  END_VAR

            L_Now_MS := GVL_STATUS.G_System_Time_MS;
L_Commit_Valid := TRUE;
L_Error_Code := 0;
L_Error_Text := '';

GVL_DISTRIBUTED_COMMIT.Peer_Commit_Ack_Expired := FALSE;
GVL_DISTRIBUTED_COMMIT.Peer_Commit_Mismatch := FALSE;
GVL_DISTRIBUTED_COMMIT.Peer_Commit_Replay_Detected := FALSE;
GVL_DISTRIBUTED_COMMIT.Peer_Commit_Missing := FALSE;
GVL_DISTRIBUTED_COMMIT.Commit_Lease_Expired := FALSE;

// Finalized publication/convergence authority.
L_Publication_Authority_Allowed :=
    GVL_Distributed_Execution_Gates.G_Runtime_Valid
    AND GVL_Distributed_Execution_Gates.G_Can_Replicate
    AND GVL_Distributed_Execution_Gates.G_Can_Own_Projection
    AND GVL_CONVERGENCE.Convergence_Lease_OK
    AND GVL_CONVERGENCE.Convergence_Release_Allowed
    AND GVL_RECOVERY_GOVERNANCE.Recovery_Governance_Valid
    AND NOT GVL_RECOVERY_GOVERNANCE.Recovery_Quarantine_Active;

GVL_DISTRIBUTED_COMMIT.Local_Publication_Commit_Epoch := GVL_DISTRIBUTED_SNAPSHOT.Distributed_Snapshot_Epoch;
GVL_DISTRIBUTED_COMMIT.Local_Prepare_Epoch := GVL_DISTRIBUTED_SNAPSHOT.Distributed_Snapshot_Epoch;

IF NOT L_Publication_Authority_Allowed THEN

    L_Commit_Valid := FALSE;

    L_Error_Code := 14999;
    L_Error_Text :=
        'Distributed publication authority restricted';

END_IF;

IF L_Commit_Valid THEN

    IF GVL_DISTRIBUTED_SNAPSHOT.Distributed_Publication_Reconciled
    AND GVL_DISTRIBUTED_SNAPSHOT.Distributed_Publication_Freeze_Valid
    AND GVL_DISTRIBUTED_SNAPSHOT.Distributed_Snapshot_Consistent
    THEN
        GVL_DISTRIBUTED_COMMIT.Publication_Prepare_Active := TRUE;
        GVL_DISTRIBUTED_COMMIT.Publication_Prepare_Valid := TRUE;
    ELSE
        GVL_DISTRIBUTED_COMMIT.Publication_Prepare_Active := FALSE;
        GVL_DISTRIBUTED_COMMIT.Publication_Prepare_Valid := FALSE;

        L_Commit_Valid := FALSE;
        L_Error_Code := 15000;
        L_Error_Text := 'Distributed immutable publication prepare invalid';
    END_IF;

END_IF;

IF GVL_DISTRIBUTED_COMMIT.Peer_Publication_Commit_Epoch > 0 THEN
    L_Peer_Session_Active := TRUE;
END_IF;

IF GVL_DISTRIBUTED_COMMIT.Peer_Prepare_Epoch > 0 THEN
    L_Peer_Session_Active := TRUE;
END_IF;

IF GVL_DISTRIBUTED_COMMIT.Peer_Commit_Ack_Valid THEN
    L_Peer_Session_Active := TRUE;
END_IF;

IF L_Commit_Valid AND L_Peer_Session_Active THEN
    L_Delta_MS := L_Now_MS - GVL_DISTRIBUTED_COMMIT.Peer_Commit_Last_Refresh_MS;

    IF GVL_DISTRIBUTED_COMMIT.Commit_Lease_Active THEN
        IF L_Delta_MS > GVL_DISTRIBUTED_COMMIT.Commit_Timeout_MS THEN
            GVL_DISTRIBUTED_COMMIT.Commit_Lease_Expired := TRUE;

            L_Commit_Valid := FALSE;
            L_Error_Code := 15001;
            L_Error_Text := 'Distributed commit lease expired';
        END_IF;
    END_IF;
END_IF;

IF L_Commit_Valid AND L_Peer_Session_Active THEN
    IF NOT GVL_DISTRIBUTED_COMMIT.Peer_Commit_Ack_Valid THEN
        GVL_DISTRIBUTED_COMMIT.Peer_Commit_Missing := TRUE;

        L_Commit_Valid := FALSE;
        L_Error_Code := 15002;
        L_Error_Text := 'Peer commit acknowledgement missing';
    END_IF;
END_IF;

IF L_Commit_Valid AND L_Peer_Session_Active THEN
    IF GVL_DISTRIBUTED_COMMIT.Peer_Publication_Commit_Epoch < GVL_DISTRIBUTED_COMMIT.Local_Publication_Commit_Epoch THEN
        GVL_DISTRIBUTED_COMMIT.Peer_Commit_Mismatch := TRUE;

        L_Commit_Valid := FALSE;
        L_Error_Code := 15003;
        L_Error_Text := 'Peer commit epoch mismatch';
    END_IF;
END_IF;

IF L_Commit_Valid AND L_Peer_Session_Active THEN
    IF GVL_DISTRIBUTED_COMMIT.Peer_Prepare_Epoch < GVL_DISTRIBUTED_COMMIT.Local_Prepare_Epoch THEN
        GVL_DISTRIBUTED_COMMIT.Peer_Commit_Replay_Detected := TRUE;

        L_Commit_Valid := FALSE;
        L_Error_Code := 15004;
        L_Error_Text := 'Peer commit replay detected';
    END_IF;
END_IF;

IF L_Commit_Valid THEN
    GVL_DISTRIBUTED_COMMIT.Distributed_Commit_Epoch := GVL_DISTRIBUTED_COMMIT.Distributed_Commit_Epoch + 1;
    GVL_DISTRIBUTED_COMMIT.Distributed_Commit_Reconciliation_Epoch := GVL_DISTRIBUTED_COMMIT.Distributed_Commit_Reconciliation_Epoch + 1;

    GVL_DISTRIBUTED_COMMIT.Publication_Commit_Requested := TRUE;

    IF L_Peer_Session_Active THEN
        GVL_DISTRIBUTED_COMMIT.Publication_Commit_Confirmed := TRUE;
        GVL_DISTRIBUTED_COMMIT.Commit_Lease_Active := TRUE;
    ELSE
        GVL_DISTRIBUTED_COMMIT.Publication_Commit_Confirmed := FALSE;
        GVL_DISTRIBUTED_COMMIT.Commit_Lease_Active := FALSE;
    END_IF;

    GVL_DISTRIBUTED_COMMIT.Distributed_Commit_Valid := TRUE;

    IF GVL_CONVERGENCE.Convergence_Release_Allowed THEN
        GVL_DISTRIBUTED_COMMIT.Distributed_Commit_Quarantine_Active := FALSE;
    END_IF;

    GVL_DISTRIBUTED_COMMIT.Commit_Last_Reconciliation_MS := L_Now_MS;

    GVL_DISTRIBUTED_COMMIT.Distributed_Commit_Last_Error_Code := 0;
    GVL_DISTRIBUTED_COMMIT.Distributed_Commit_Last_Error_Text := '';
ELSE
    GVL_DISTRIBUTED_COMMIT.Publication_Commit_Confirmed := FALSE;

    GVL_DISTRIBUTED_COMMIT.Distributed_Commit_Valid := FALSE;
    GVL_DISTRIBUTED_COMMIT.Distributed_Commit_Quarantine_Active := TRUE;

    GVL_DISTRIBUTED_COMMIT.Distributed_Commit_Last_Error_Code := L_Error_Code;
    GVL_DISTRIBUTED_COMMIT.Distributed_Commit_Last_Error_Text := L_Error_Text;
END_IF;
          
END_PROGRAM

PROGRAM PRG_Execution_Progress_Causality_Governor

            IF GVL_PHYSICAL_DEADLOCK_RESOLUTION_FABRIC.Physical_Deadlock_Resolution_Granted
AND NOT GVL_EXECUTION_PROGRESS_CAUSALITY_FABRIC.Distributed_Execution_Stall_Detected
AND NOT GVL_EXECUTION_PROGRESS_CAUSALITY_FABRIC.Execution_Progress_Divergence_Detected
AND NOT GVL_EXECUTION_PROGRESS_CAUSALITY_FABRIC.Recovery_Progress_Oscillation_Detected THEN

    GVL_EXECUTION_PROGRESS_CAUSALITY_FABRIC.Execution_Progress_Causality_Valid := TRUE;
    GVL_EXECUTION_PROGRESS_CAUSALITY_FABRIC.Execution_Progress_Causality_Granted := TRUE;
    GVL_EXECUTION_PROGRESS_CAUSALITY_FABRIC.Progress_Causality_Grounded := TRUE;
    GVL_EXECUTION_PROGRESS_CAUSALITY_FABRIC.Deterministic_Execution_Continuation_Valid := TRUE;
END_IF;
          
END_PROGRAM

PROGRAM PRG_Safety_Observability_Truth_Governor

            IF GVL_DISTRIBUTED_FORWARD_PROGRESS_FABRIC.Distributed_Forward_Progress_Granted
AND NOT GVL_SAFETY_OBSERVABILITY_TRUTH_FABRIC.FakeSafe_Projection_Detected
AND NOT GVL_SAFETY_OBSERVABILITY_TRUTH_FABRIC.Telemetry_Reality_Divergence_Detected
AND NOT GVL_SAFETY_OBSERVABILITY_TRUTH_FABRIC.Stale_Safety_Projection_Detected
AND NOT GVL_SAFETY_OBSERVABILITY_TRUTH_FABRIC.Safety_Observability_Fork_Detected THEN

    GVL_SAFETY_OBSERVABILITY_TRUTH_FABRIC.Safety_Observability_Truth_Valid := TRUE;
    GVL_SAFETY_OBSERVABILITY_TRUTH_FABRIC.Safety_Observability_Truth_Granted := TRUE;
    GVL_SAFETY_OBSERVABILITY_TRUTH_FABRIC.Safety_Reality_Projection_Valid := TRUE;
    GVL_SAFETY_OBSERVABILITY_TRUTH_FABRIC.Observability_Reality_Equivalence_Granted := TRUE;
    GVL_SAFETY_OBSERVABILITY_TRUTH_FABRIC.Physical_Safety_Projection_Canonical := TRUE;
END_IF;
          
END_PROGRAM

PROGRAM PRG_System_Trend
  VAR
    fbTrendLogger : FB_Trend_Logger;
    fbTrendAdapter : FB_Trend_Adapter;
    L_TrendConfig : ST_Trend_Config;
    L_TrendData : ST_Trend_Data;
    L_Average : REAL;
    L_Min : REAL;
    L_Max : REAL;
    L_Trend_Up : BOOL;
    L_Trend_Down : BOOL;
  END_VAR

            // Minimal production trend channel: room temperature 1.
L_TrendConfig.enabled := TRUE;
L_TrendConfig.param_type := 1;
L_TrendConfig.zone_id := 1;
L_TrendConfig.deviation_threshold_percent := REAL#1.0;
L_TrendConfig.history_days := 7;

